KUKA KRL program: f1_Kuka_APT218T02S18.SRC

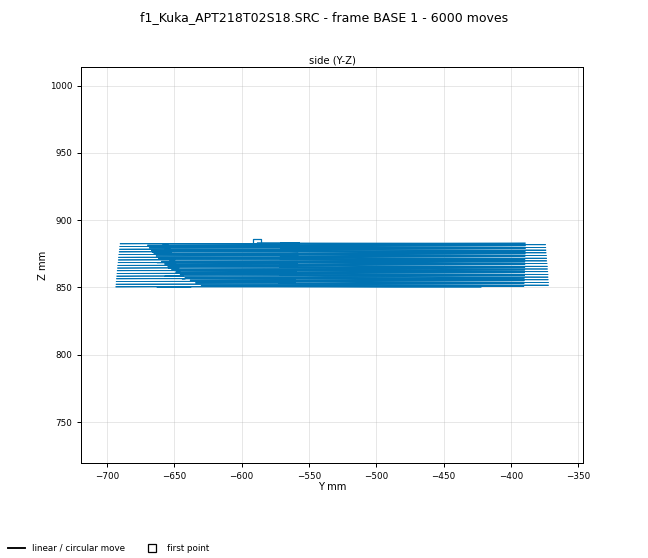
[picture p0: tool path of f1_Kuka_APT218T02S18.SRC in frame BASE 1, 6000 of 6001 moves have a stored position in this frame; points joined in program order, loops and branches not executed]
&ACCESS RVP
&REL 2
&PARAM TEMPLATE = C:\KRC\Roboter\Template\vorgabe
&PARAM EDITMASK = *
DEF f1_Kuka_APT218T02S18()


;FOLD INI;%{PE}%V3.2.0,%MKUKATPBASIS,%CINIT,%VCOMMON,%P
  ;FOLD BAS INI;%{E}%V3.2.0,%MKUKATPBASIS,%CINIT,%VINIT,%P
    GLOBAL INTERRUPT DECL 3 WHEN $STOPMESS==TRUE DO IR_STOPM ( )
    INTERRUPT ON 3
    BAS (#INITMOV,0 )
  ;ENDFOLD (BAS INI)
  ;FOLD USER INI;%{E}%V3.2.0,%MKUKATPUSER,%CINIT,%VINIT,%P
    ;Make your modifications here
  ;ENDFOLD (USER INI)
;ENDFOLD (INI)


;*** Make Null PTP Move
  PTP $pos_act

;*** Auto Load The Correct TOOL Data
  $tool=tool_data[2]

;*** Auto Load The Correct BASE Data
  $base=base_data[1]

  $ADVANCE = 5

;*** Restate Last Velocity
MMPM(30000.0)
SetRPM(8000)
LIN {X 0.122,Y -588.379,Z 883.406,A 0.000,B 0.000,C 90.000,E1 109.033} C_DIS
LIN {X -0.101,Y -579.806,Z 883.404,A 0.000,B 0.000,C 90.000,E1 108.671} C_DIS
LIN {X -0.188,Y -568.248,Z 883.402,A 0.000,B 0.000,C 90.000,E1 108.290} C_DIS
LIN {X -0.241,Y -564.785,Z 883.401,A 0.000,B 0.000,C 90.000,E1 108.181} C_DIS
LIN {X -0.107,Y -562.267,Z 883.400,A 0.000,B 0.000,C 90.000,E1 108.055} C_DIS
LIN {X 0.277,Y -559.252,Z 883.399,A 0.000,B 0.000,C 90.000,E1 107.819} C_DIS
LIN {X 0.169,Y -557.826,Z 883.398,A 0.000,B 0.000,C 90.000,E1 107.583} C_DIS
LIN {X -0.019,Y -557.157,Z 883.396,A 0.000,B 0.000,C 90.000,E1 107.221} C_DIS
LIN {X -0.140,Y -557.033,Z 883.393,A 0.000,B 0.000,C 90.000,E1 106.677} C_DIS
LIN {X 0.137,Y -558.022,Z 883.376,A 0.000,B 0.000,C 90.000,E1 103.592} C_DIS
LIN {X 0.043,Y -559.152,Z 883.365,A 0.000,B 0.000,C 90.000,E1 101.658} C_DIS
LIN {X -0.031,Y -560.530,Z 883.354,A 0.000,B 0.000,C 90.000,E1 99.726} C_DIS
LIN {X -0.015,Y -561.492,Z 883.346,A 0.000,B 0.000,C 90.000,E1 98.341} C_DIS
LIN {X 0.100,Y -562.358,Z 883.339,A 0.000,B 0.000,C 90.000,E1 96.947} C_DIS
LIN {X 0.092,Y -563.149,Z 883.331,A 0.000,B 0.000,C 90.000,E1 95.568} C_DIS
LIN {X 0.246,Y -563.909,Z 883.322,A 0.000,B 0.000,C 90.000,E1 93.898} C_DIS
LIN {X 0.231,Y -564.401,Z 883.314,A 0.000,B 0.000,C 90.000,E1 92.522} C_DIS
LIN {X -0.229,Y -564.932,Z 883.305,A 0.000,B 0.000,C 90.000,E1 90.917} C_DIS
LIN {X -0.237,Y -565.272,Z 883.297,A 0.000,B 0.000,C 90.000,E1 89.542} C_DIS
LIN {X -0.226,Y -565.571,Z 883.290,A 0.000,B 0.000,C 90.000,E1 88.165} C_DIS
LIN {X -0.093,Y -565.844,Z 883.281,A 0.000,B 0.000,C 90.000,E1 86.502} C_DIS
LIN {X -0.033,Y -566.089,Z 883.273,A 0.000,B 0.000,C 90.000,E1 85.122} C_DIS
LIN {X -0.274,Y -566.409,Z 883.262,A 0.000,B 0.000,C 90.000,E1 83.223} C_DIS
LIN {X -0.283,Y -566.973,Z 883.250,A 0.000,B 0.000,C 90.000,E1 81.027} C_DIS
LIN {X 0.107,Y -567.557,Z 883.241,A 0.000,B 0.000,C 90.000,E1 79.342} C_DIS
LIN {X 0.241,Y -568.440,Z 883.230,A 0.000,B 0.000,C 90.000,E1 77.409} C_DIS
LIN {X 0.029,Y -569.048,Z 883.223,A 0.000,B 0.000,C 90.000,E1 76.061} C_DIS
LIN {X -0.040,Y -569.635,Z 883.215,A 0.000,B 0.000,C 90.000,E1 74.700} C_DIS
LIN {X -0.120,Y -570.012,Z 883.209,A 0.000,B 0.000,C 90.000,E1 73.614} C_DIS
LIN {X 0.162,Y -570.430,Z 883.200,A 0.000,B 0.000,C 90.000,E1 71.945} C_DIS
LIN {X 0.102,Y -570.623,Z 883.194,A 0.000,B 0.000,C 90.000,E1 70.859} C_DIS
LIN {X 0.237,Y -570.806,Z 883.188,A 0.000,B 0.000,C 90.000,E1 69.752} C_DIS
LIN {X -0.001,Y -570.993,Z 883.176,A 0.000,B 0.000,C 90.000,E1 67.592} C_DIS
LIN {X 0.141,Y -571.068,Z 883.169,A 0.000,B 0.000,C 90.000,E1 66.485} C_DIS
LIN {X 0.169,Y -571.046,Z 883.160,A 0.000,B 0.000,C 90.000,E1 64.845} C_DIS
LIN {X 0.190,Y -570.924,Z 883.151,A 0.000,B 0.000,C 90.000,E1 63.204} C_DIS
LIN {X -0.057,Y -570.579,Z 883.142,A 0.000,B 0.000,C 90.000,E1 61.591} C_DIS
LIN {X 0.309,Y -570.340,Z 883.136,A 0.000,B 0.000,C 90.000,E1 60.461} C_DIS
LIN {X 0.073,Y -570.058,Z 883.132,A 0.000,B 0.000,C 90.000,E1 59.665} C_DIS
LIN {X -0.113,Y -569.130,Z 883.122,A 0.000,B 0.000,C 90.000,E1 58.043} C_DIS
LIN {X 0.113,Y -568.574,Z 883.118,A 0.000,B 0.000,C 90.000,E1 57.199} C_DIS
LIN {X 0.155,Y -567.877,Z 883.113,A 0.000,B 0.000,C 90.000,E1 56.373} C_DIS
LIN {X -0.158,Y -566.857,Z 883.107,A 0.000,B 0.000,C 90.000,E1 55.308} C_DIS
LIN {X -0.016,Y -565.616,Z 883.101,A 0.000,B 0.000,C 90.000,E1 54.196} C_DIS
LIN {X -0.352,Y -564.093,Z 883.095,A 0.000,B 0.000,C 90.000,E1 53.130} C_DIS
LIN {X -0.028,Y -562.837,Z 883.090,A 0.000,B 0.000,C 90.000,E1 52.271} C_DIS
LIN {X -0.161,Y -561.473,Z 883.086,A 0.000,B 0.000,C 90.000,E1 51.457} C_DIS
LIN {X 0.127,Y -559.875,Z 883.081,A 0.000,B 0.000,C 90.000,E1 50.598} C_DIS
LIN {X -0.124,Y -558.727,Z 883.078,A 0.000,B 0.000,C 90.000,E1 50.070} C_DIS
LIN {X 0.061,Y -556.766,Z 883.074,A 0.000,B 0.000,C 90.000,E1 49.218} C_DIS
LIN {X 0.296,Y -553.482,Z 883.067,A 0.000,B 0.000,C 90.000,E1 48.081} C_DIS
LIN {X 0.004,Y -551.691,Z 883.064,A 0.000,B 0.000,C 90.000,E1 47.553} C_DIS
LIN {X 0.113,Y -548.706,Z 883.060,A 0.000,B 0.000,C 90.000,E1 46.701} C_DIS
LIN {X -0.205,Y -545.511,Z 883.055,A 0.000,B 0.000,C 90.000,E1 45.891} C_DIS
LIN {X 0.217,Y -541.967,Z 883.050,A 0.000,B 0.000,C 90.000,E1 45.000} C_DIS
LIN {X 0.018,Y -538.556,Z 883.046,A 0.000,B 0.000,C 90.000,E1 44.312} C_DIS
LIN {X -0.203,Y -534.722,Z 883.042,A 0.000,B 0.000,C 90.000,E1 43.623} C_DIS
LIN {X -0.090,Y -530.576,Z 883.038,A 0.000,B 0.000,C 90.000,E1 42.894} C_DIS
LIN {X 0.211,Y -527.049,Z 883.035,A 0.000,B 0.000,C 90.000,E1 42.285} C_DIS
LIN {X 0.045,Y -521.421,Z 883.030,A 0.000,B 0.000,C 90.000,E1 41.434} C_DIS
LIN {X 0.007,Y -513.993,Z 883.025,A 0.000,B 0.000,C 90.000,E1 40.415} C_DIS
LIN {X 0.301,Y -508.245,Z 883.021,A 0.000,B 0.000,C 90.000,E1 39.644} C_DIS
LIN {X 0.213,Y -501.947,Z 883.016,A 0.000,B 0.000,C 90.000,E1 38.910} C_DIS
LIN {X 0.220,Y -497.947,Z 883.014,A 0.000,B 0.000,C 90.000,E1 38.463} C_DIS
LIN {X -0.149,Y -489.660,Z 883.009,A 0.000,B 0.000,C 90.000,E1 37.649} C_DIS
LIN {X -0.010,Y -483.974,Z 883.006,A 0.000,B 0.000,C 90.000,E1 37.076} C_DIS
LIN {X 0.171,Y -476.519,Z 883.002,A 0.000,B 0.000,C 90.000,E1 36.377} C_DIS
LIN {X -0.193,Y -466.025,Z 882.997,A 0.000,B 0.000,C 90.000,E1 35.518} C_DIS
LIN {X -0.045,Y -458.299,Z 882.994,A 0.000,B 0.000,C 90.000,E1 34.865} C_DIS
LIN {X -0.104,Y -450.565,Z 882.990,A 0.000,B 0.000,C 90.000,E1 34.246} C_DIS
LIN {X 0.184,Y -435.026,Z 882.983,A 0.000,B 0.000,C 90.000,E1 32.959} C_DIS
LIN {X -0.153,Y -418.321,Z 882.975,A 0.000,B 0.000,C 90.000,E1 31.592} C_DIS
LIN {X -0.172,Y -404.709,Z 882.968,A 0.000,B 0.000,C 90.000,E1 30.335} C_DIS
LIN {X 0.006,Y -397.858,Z 882.964,A 0.000,B 0.000,C 90.000,E1 29.589} C_DIS
LIN {X -0.089,Y -395.270,Z 882.963,A 0.000,B 0.000,C 90.000,E1 29.283} C_DIS
LIN {X 0.077,Y -393.465,Z 882.961,A 0.000,B 0.000,C 90.000,E1 28.999} C_DIS
LIN {X 0.060,Y -391.088,Z 882.958,A 0.000,B 0.000,C 90.000,E1 28.487} C_DIS
LIN {X -0.130,Y -390.109,Z 882.956,A 0.000,B 0.000,C 90.000,E1 28.153} C_DIS
LIN {X -0.125,Y -389.776,Z 882.955,A 0.000,B 0.000,C 90.000,E1 27.975} C_DIS
LIN {X -0.066,Y -389.241,Z 882.952,A 0.000,B 0.000,C 90.000,E1 27.436} C_DIS
LIN {X -0.178,Y -389.129,Z 882.948,A 0.000,B 0.000,C 90.000,E1 26.744} C_DIS
LIN {X -0.114,Y -390.003,Z 882.939,A 0.000,B 0.000,C 90.000,E1 24.951} C_DIS
LIN {X 0.108,Y -392.719,Z 882.921,A 0.000,B 0.000,C 90.000,E1 21.716} C_DIS
LIN {X -0.171,Y -394.920,Z 882.909,A 0.000,B 0.000,C 90.000,E1 19.631} C_DIS
LIN {X -0.095,Y -397.735,Z 882.895,A 0.000,B 0.000,C 90.000,E1 17.149} C_DIS
LIN {X 0.184,Y -401.298,Z 882.880,A 0.000,B 0.000,C 90.000,E1 14.300} C_DIS
LIN {X -0.001,Y -405.149,Z 882.864,A 0.000,B 0.000,C 90.000,E1 11.535} C_DIS
LIN {X 0.084,Y -408.893,Z 882.851,A 0.000,B 0.000,C 90.000,E1 9.095} C_DIS
LIN {X -0.156,Y -413.579,Z 882.835,A 0.000,B 0.000,C 90.000,E1 6.372} C_DIS
LIN {X 0.009,Y -418.079,Z 882.822,A 0.000,B 0.000,C 90.000,E1 3.955} C_DIS
LIN {X -0.043,Y -425.252,Z 882.803,A 0.000,B 0.000,C 90.000,E1 0.573} C_DIS
LIN {X -0.010,Y -430.285,Z 882.791,A 0.000,B 0.000,C 90.000,E1 358.453} C_DIS
LIN {X -0.159,Y -437.144,Z 882.777,A 0.000,B 0.000,C 90.000,E1 355.812} C_DIS
LIN {X 0.066,Y -439.313,Z 882.773,A 0.000,B 0.000,C 90.000,E1 355.122} C_DIS
LIN {X 0.067,Y -442.262,Z 882.770,A 0.000,B 0.000,C 90.000,E1 354.546} C_DIS
LIN {X 0.180,Y -444.846,Z 882.768,A 0.000,B 0.000,C 90.000,E1 354.204} C_DIS
LIN {X 0.121,Y -449.563,Z 882.766,A 0.000,B 0.000,C 90.000,E1 353.856} C_DIS
LIN {X 0.062,Y -455.330,Z 882.764,A 0.000,B 0.000,C 90.000,E1 353.571} C_DIS
LIN {X -0.058,Y -468.891,Z 882.761,A 0.000,B 0.000,C 90.000,E1 352.996} C_DIS
LIN {X -0.002,Y -477.211,Z 882.759,A 0.000,B 0.000,C 90.000,E1 352.591} C_DIS
LIN {X 0.067,Y -483.618,Z 882.757,A 0.000,B 0.000,C 90.000,E1 352.243} C_DIS
LIN {X 0.101,Y -491.818,Z 882.754,A 0.000,B 0.000,C 90.000,E1 351.781} C_DIS
LIN {X 0.245,Y -501.546,Z 882.751,A 0.000,B 0.000,C 90.000,E1 351.197} C_DIS
LIN {X 0.051,Y -510.970,Z 882.748,A 0.000,B 0.000,C 90.000,E1 350.622} C_DIS
LIN {X 0.091,Y -518.862,Z 882.745,A 0.000,B 0.000,C 90.000,E1 350.095} C_DIS
LIN {X 0.016,Y -526.453,Z 882.742,A 0.000,B 0.000,C 90.000,E1 349.567} C_DIS
LIN {X 0.149,Y -532.466,Z 882.740,A 0.000,B 0.000,C 90.000,E1 349.106} C_DIS
LIN {X 0.151,Y -539.715,Z 882.736,A 0.000,B 0.000,C 90.000,E1 348.522} C_DIS
LIN {X -0.009,Y -546.525,Z 882.733,A 0.000,B 0.000,C 90.000,E1 347.937} C_DIS
LIN {X -0.075,Y -554.603,Z 882.729,A 0.000,B 0.000,C 90.000,E1 347.173} C_DIS
LIN {X -0.137,Y -561.000,Z 882.725,A 0.000,B 0.000,C 90.000,E1 346.520} C_DIS
LIN {X -0.028,Y -567.119,Z 882.721,A 0.000,B 0.000,C 90.000,E1 345.825} C_DIS
LIN {X -0.095,Y -571.726,Z 882.718,A 0.000,B 0.000,C 90.000,E1 345.283} C_DIS
LIN {X -0.175,Y -579.173,Z 882.713,A 0.000,B 0.000,C 90.000,E1 344.338} C_DIS
LIN {X 0.159,Y -584.078,Z 882.709,A 0.000,B 0.000,C 90.000,E1 343.630} C_DIS
LIN {X -0.176,Y -590.395,Z 882.704,A 0.000,B 0.000,C 90.000,E1 342.725} C_DIS
LIN {X 0.070,Y -597.021,Z 882.698,A 0.000,B 0.000,C 90.000,E1 341.638} C_DIS
LIN {X -0.155,Y -603.051,Z 882.692,A 0.000,B 0.000,C 90.000,E1 340.604} C_DIS
LIN {X -0.235,Y -607.309,Z 882.688,A 0.000,B 0.000,C 90.000,E1 339.826} C_DIS
LIN {X -0.158,Y -614.014,Z 882.681,A 0.000,B 0.000,C 90.000,E1 338.518} C_DIS
LIN {X -0.159,Y -618.460,Z 882.676,A 0.000,B 0.000,C 90.000,E1 337.614} C_DIS
LIN {X 0.116,Y -623.243,Z 882.670,A 0.000,B 0.000,C 90.000,E1 336.561} C_DIS
LIN {X 0.131,Y -627.747,Z 882.664,A 0.000,B 0.000,C 90.000,E1 335.537} C_DIS
LIN {X -0.049,Y -631.918,Z 882.659,A 0.000,B 0.000,C 90.000,E1 334.537} C_DIS
LIN {X 0.096,Y -635.794,Z 882.653,A 0.000,B 0.000,C 90.000,E1 333.512} C_DIS
LIN {X 0.293,Y -639.458,Z 882.647,A 0.000,B 0.000,C 90.000,E1 332.487} C_DIS
LIN {X 0.036,Y -643.618,Z 882.640,A 0.000,B 0.000,C 90.000,E1 331.257} C_DIS
LIN {X 0.237,Y -648.155,Z 882.632,A 0.000,B 0.000,C 90.000,E1 329.744} C_DIS
LIN {X 0.258,Y -650.302,Z 882.628,A 0.000,B 0.000,C 90.000,E1 328.997} C_DIS
LIN {X -0.065,Y -653.728,Z 882.621,A 0.000,B 0.000,C 90.000,E1 327.788} C_DIS
LIN {X 0.110,Y -656.122,Z 882.616,A 0.000,B 0.000,C 90.000,E1 326.786} C_DIS
LIN {X 0.128,Y -658.310,Z 882.610,A 0.000,B 0.000,C 90.000,E1 325.801} C_DIS
LIN {X 0.183,Y -660.174,Z 882.605,A 0.000,B 0.000,C 90.000,E1 324.815} C_DIS
LIN {X 0.265,Y -661.759,Z 882.599,A 0.000,B 0.000,C 90.000,E1 323.829} C_DIS
LIN {X 0.363,Y -663.180,Z 882.594,A 0.000,B 0.000,C 90.000,E1 322.844} C_DIS
LIN {X -0.023,Y -664.153,Z 882.590,A 0.000,B 0.000,C 90.000,E1 322.145} C_DIS
LIN {X -0.040,Y -665.507,Z 882.583,A 0.000,B 0.000,C 90.000,E1 320.928} C_DIS
LIN {X 0.065,Y -666.817,Z 882.576,A 0.000,B 0.000,C 90.000,E1 319.703} C_DIS
LIN {X 0.103,Y -668.353,Z 882.568,A 0.000,B 0.000,C 90.000,E1 318.243} C_DIS
LIN {X -0.324,Y -669.643,Z 882.561,A 0.000,B 0.000,C 90.000,E1 317.067} C_DIS
LIN {X 0.217,Y -670.951,Z 882.555,A 0.000,B 0.000,C 90.000,E1 315.810} C_DIS
LIN {X 0.299,Y -672.265,Z 882.548,A 0.000,B 0.000,C 90.000,E1 314.595} C_DIS
LIN {X -0.022,Y -673.927,Z 882.539,A 0.000,B 0.000,C 90.000,E1 312.933} C_DIS
LIN {X -0.363,Y -675.092,Z 882.532,A 0.000,B 0.000,C 90.000,E1 311.757} C_DIS
LIN {X -0.208,Y -675.929,Z 882.526,A 0.000,B 0.000,C 90.000,E1 310.782} C_DIS
LIN {X 0.118,Y -677.365,Z 882.517,A 0.000,B 0.000,C 90.000,E1 309.072} C_DIS
LIN {X -0.084,Y -678.489,Z 882.509,A 0.000,B 0.000,C 90.000,E1 307.649} C_DIS
LIN {X -0.163,Y -679.400,Z 882.503,A 0.000,B 0.000,C 90.000,E1 306.457} C_DIS
LIN {X 0.172,Y -680.053,Z 882.497,A 0.000,B 0.000,C 90.000,E1 305.471} C_DIS
LIN {X 0.303,Y -681.034,Z 882.488,A 0.000,B 0.000,C 90.000,E1 303.785} C_DIS
LIN {X 0.448,Y -681.993,Z 882.480,A 0.000,B 0.000,C 90.000,E1 302.339} C_DIS
LIN {X 0.060,Y -683.481,Z 882.469,A 0.000,B 0.000,C 90.000,E1 300.463} C_DIS
LIN {X 0.181,Y -685.412,Z 882.457,A 0.000,B 0.000,C 90.000,E1 298.309} C_DIS
LIN {X 0.129,Y -687.513,Z 882.447,A 0.000,B 0.000,C 90.000,E1 296.411} C_DIS
LIN {X 0.345,Y -688.947,Z 882.440,A 0.000,B 0.000,C 90.000,E1 295.207} C_DIS
LIN {X 0.069,Y -689.832,Z 882.435,A 0.000,B 0.000,C 90.000,E1 294.283} C_DIS
LIN {X 0.135,Y -690.317,Z 882.431,A 0.000,B 0.000,C 90.000,E1 293.567} C_DIS
LIN {X 0.092,Y -690.368,Z 882.430,A 0.000,B 0.000,C 90.000,E1 293.334} C_DIS
LIN {X -0.350,Y -690.024,Z 882.427,A 0.000,B 0.000,C 90.000,E1 292.898} C_DIS
LIN {X -0.120,Y -689.571,Z 882.426,A 0.000,B 0.000,C 90.000,E1 292.642} C_DIS
LIN {X 0.072,Y -687.982,Z 882.423,A 0.000,B 0.000,C 90.000,E1 292.153} C_DIS
LIN {X 0.183,Y -687.443,Z 882.422,A 0.000,B 0.000,C 90.000,E1 292.025} C_DIS
LIN {X 0.294,Y -686.610,Z 882.422,A 0.000,B 0.000,C 90.000,E1 291.897} C_DIS
LIN {X 0.254,Y -684.050,Z 882.421,A 0.000,B 0.000,C 90.000,E1 291.663} C_DIS
LIN {X -0.185,Y -682.758,Z 882.420,A 0.000,B 0.000,C 90.000,E1 291.589} C_DIS
LIN {X 0.055,Y -679.828,Z 882.419,A 0.000,B 0.000,C 90.000,E1 291.354} C_DIS
LIN {X -0.284,Y -677.735,Z 882.418,A 0.000,B 0.000,C 90.000,E1 291.280} C_DIS
LIN {X 0.307,Y -669.422,Z 882.417,A 0.000,B 0.000,C 90.000,E1 290.972} C_DIS
LIN {X 0.039,Y -661.806,Z 882.416,A 0.000,B 0.000,C 90.000,E1 290.791} C_DIS
LIN {X -0.137,Y -660.012,Z 882.415,A 0.000,B 0.000,C 90.000,E1 290.737} C_DIS
LIN {X -0.188,Y -655.626,Z 882.414,A 0.000,B 0.000,C 90.000,E1 290.536} C_DIS
LIN {X 0.371,Y -655.532,Z 882.414,A 0.000,B 0.000,C 90.000,E1 290.482} C_DIS
LIN {X -0.298,Y -654.580,Z 882.413,A 0.000,B 0.000,C 90.000,E1 290.429} C_DIS
LIN {X -0.342,Y -654.560,Z 882.413,A 0.000,B 0.000,C 90.000,E1 290.429} C_DIS
LIN {X 0.106,Y -654.455,Z 882.412,A 0.000,B 0.000,C 90.000,E1 290.174} C_DIS
LIN {X -0.068,Y -655.646,Z 882.410,A 0.000,B 0.000,C 90.000,E1 289.758} C_DIS
LIN {X 0.128,Y -658.793,Z 882.406,A 0.000,B 0.000,C 90.000,E1 289.087} C_DIS
LIN {X 0.056,Y -665.349,Z 882.399,A 0.000,B 0.000,C 90.000,E1 287.873} C_DIS
LIN {X -0.010,Y -668.755,Z 882.395,A 0.000,B 0.000,C 90.000,E1 287.149} C_DIS
LIN {X -0.238,Y -671.708,Z 882.391,A 0.000,B 0.000,C 90.000,E1 286.441} C_DIS
LIN {X -0.184,Y -673.408,Z 882.389,A 0.000,B 0.000,C 90.000,E1 285.953} C_DIS
LIN {X 0.287,Y -675.387,Z 882.385,A 0.000,B 0.000,C 90.000,E1 285.190} C_DIS
LIN {X 0.134,Y -676.960,Z 882.381,A 0.000,B 0.000,C 90.000,E1 284.481} C_DIS
LIN {X -0.003,Y -678.229,Z 882.377,A 0.000,B 0.000,C 90.000,E1 283.772} C_DIS
LIN {X -0.129,Y -679.262,Z 882.373,A 0.000,B 0.000,C 90.000,E1 283.063} C_DIS
LIN {X -0.249,Y -679.961,Z 882.369,A 0.000,B 0.000,C 90.000,E1 282.355} C_DIS
LIN {X 0.338,Y -680.308,Z 882.366,A 0.000,B 0.000,C 90.000,E1 281.827} C_DIS
LIN {X 0.125,Y -680.466,Z 882.363,A 0.000,B 0.000,C 90.000,E1 281.366} C_DIS
LIN {X 0.008,Y -680.140,Z 882.359,A 0.000,B 0.000,C 90.000,E1 280.658} C_DIS
LIN {X -0.199,Y -679.695,Z 882.357,A 0.000,B 0.000,C 90.000,E1 280.197} C_DIS
LIN {X -0.287,Y -678.957,Z 882.354,A 0.000,B 0.000,C 90.000,E1 279.726} C_DIS
LIN {X 0.173,Y -677.860,Z 882.351,A 0.000,B 0.000,C 90.000,E1 279.208} C_DIS
LIN {X -0.038,Y -676.482,Z 882.349,A 0.000,B 0.000,C 90.000,E1 278.746} C_DIS
LIN {X -0.096,Y -675.722,Z 882.347,A 0.000,B 0.000,C 90.000,E1 278.511} C_DIS
LIN {X -0.318,Y -673.947,Z 882.345,A 0.000,B 0.000,C 90.000,E1 278.049} C_DIS
LIN {X 0.118,Y -671.850,Z 882.342,A 0.000,B 0.000,C 90.000,E1 277.530} C_DIS
LIN {X -0.126,Y -668.852,Z 882.339,A 0.000,B 0.000,C 90.000,E1 276.947} C_DIS
LIN {X 0.181,Y -665.352,Z 882.335,A 0.000,B 0.000,C 90.000,E1 276.315} C_DIS
LIN {X -0.108,Y -662.244,Z 882.333,A 0.000,B 0.000,C 90.000,E1 275.853} C_DIS
LIN {X 0.239,Y -658.650,Z 882.330,A 0.000,B 0.000,C 90.000,E1 275.334} C_DIS
LIN {X -0.197,Y -653.477,Z 882.326,A 0.000,B 0.000,C 90.000,E1 274.759} C_DIS
LIN {X 0.058,Y -648.780,Z 882.324,A 0.000,B 0.000,C 90.000,E1 274.245} C_DIS
LIN {X -0.202,Y -643.723,Z 882.321,A 0.000,B 0.000,C 90.000,E1 273.784} C_DIS
LIN {X 0.298,Y -637.049,Z 882.318,A 0.000,B 0.000,C 90.000,E1 273.154} C_DIS
LIN {X -0.158,Y -631.515,Z 882.315,A 0.000,B 0.000,C 90.000,E1 272.751} C_DIS
LIN {X -0.289,Y -623.990,Z 882.312,A 0.000,B 0.000,C 90.000,E1 272.236} C_DIS
LIN {X -0.088,Y -617.778,Z 882.310,A 0.000,B 0.000,C 90.000,E1 271.835} C_DIS
LIN {X -0.203,Y -611.264,Z 882.308,A 0.000,B 0.000,C 90.000,E1 271.489} C_DIS
LIN {X -0.011,Y -604.489,Z 882.306,A 0.000,B 0.000,C 90.000,E1 271.146} C_DIS
LIN {X -0.109,Y -597.612,Z 882.305,A 0.000,B 0.000,C 90.000,E1 270.859} C_DIS
LIN {X 0.162,Y -590.393,Z 882.303,A 0.000,B 0.000,C 90.000,E1 270.573} C_DIS
LIN {X -0.278,Y -582.943,Z 882.302,A 0.000,B 0.000,C 90.000,E1 270.401} C_DIS
LIN {X 0.038,Y -577.504,Z 882.301,A 0.000,B 0.000,C 90.000,E1 270.229} C_DIS
LIN {X -0.107,Y -571.034,Z 882.301,A 0.000,B 0.000,C 90.000,E1 270.115} C_DIS
LIN {X 0.195,Y -563.729,Z 882.300,A 0.000,B 0.000,C 90.000,E1 270.000} C_DIS
LIN {X -0.009,Y -552.379,Z 882.300,A 0.000,B 0.000,C 90.000,E1 269.943} C_DIS
LIN {X -0.195,Y -549.486,Z 882.299,A 0.000,B 0.000,C 90.000,E1 269.885} C_DIS
LIN {X -0.224,Y -549.437,Z 882.299,A 0.000,B 0.000,C 90.000,E1 269.885} C_DIS
LIN {X 0.068,Y -546.726,Z 882.298,A 0.000,B 0.000,C 90.000,E1 269.542} C_DIS
LIN {X -0.056,Y -546.333,Z 882.297,A 0.000,B 0.000,C 90.000,E1 269.484} C_DIS
LIN {X 0.115,Y -545.774,Z 882.296,A 0.000,B 0.000,C 90.000,E1 269.255} C_DIS
LIN {X -0.249,Y -544.841,Z 882.293,A 0.000,B 0.000,C 90.000,E1 268.740} C_DIS
LIN {X 0.254,Y -541.460,Z 882.271,A 0.000,B 0.000,C 90.000,E1 264.723} C_DIS
LIN {X -0.067,Y -540.539,Z 882.263,A 0.000,B 0.000,C 90.000,E1 263.337} C_DIS
LIN {X 0.066,Y -539.640,Z 882.257,A 0.000,B 0.000,C 90.000,E1 262.186} C_DIS
LIN {X -0.210,Y -538.259,Z 882.249,A 0.000,B 0.000,C 90.000,E1 260.792} C_DIS
LIN {X 0.080,Y -536.471,Z 882.239,A 0.000,B 0.000,C 90.000,E1 259.050} C_DIS
LIN {X -0.153,Y -534.963,Z 882.231,A 0.000,B 0.000,C 90.000,E1 257.645} C_DIS
LIN {X 0.177,Y -533.606,Z 882.225,A 0.000,B 0.000,C 90.000,E1 256.464} C_DIS
LIN {X 0.052,Y -531.429,Z 882.215,A 0.000,B 0.000,C 90.000,E1 254.755} C_DIS
LIN {X 0.164,Y -529.324,Z 882.206,A 0.000,B 0.000,C 90.000,E1 253.015} C_DIS
LIN {X 0.059,Y -527.638,Z 882.198,A 0.000,B 0.000,C 90.000,E1 251.583} C_DIS
LIN {X -0.248,Y -525.386,Z 882.188,A 0.000,B 0.000,C 90.000,E1 249.880} C_DIS
LIN {X -0.090,Y -523.463,Z 882.180,A 0.000,B 0.000,C 90.000,E1 248.411} C_DIS
LIN {X 0.222,Y -521.303,Z 882.172,A 0.000,B 0.000,C 90.000,E1 246.922} C_DIS
LIN {X -0.129,Y -519.547,Z 882.165,A 0.000,B 0.000,C 90.000,E1 245.793} C_DIS
LIN {X -0.148,Y -517.318,Z 882.157,A 0.000,B 0.000,C 90.000,E1 244.332} C_DIS
LIN {X 0.006,Y -515.924,Z 882.152,A 0.000,B 0.000,C 90.000,E1 243.435} C_DIS
LIN {X -0.198,Y -513.885,Z 882.146,A 0.000,B 0.000,C 90.000,E1 242.281} C_DIS
LIN {X -0.095,Y -511.318,Z 882.138,A 0.000,B 0.000,C 90.000,E1 240.795} C_DIS
LIN {X -0.237,Y -508.789,Z 882.130,A 0.000,B 0.000,C 90.000,E1 239.331} C_DIS
LIN {X -0.051,Y -506.637,Z 882.123,A 0.000,B 0.000,C 90.000,E1 238.122} C_DIS
LIN {X -0.216,Y -504.969,Z 882.118,A 0.000,B 0.000,C 90.000,E1 237.248} C_DIS
LIN {X 0.182,Y -502.556,Z 882.111,A 0.000,B 0.000,C 90.000,E1 236.008} C_DIS
LIN {X 0.247,Y -500.622,Z 882.106,A 0.000,B 0.000,C 90.000,E1 235.102} C_DIS
LIN {X -0.227,Y -495.716,Z 882.095,A 0.000,B 0.000,C 90.000,E1 233.050} C_DIS
LIN {X -0.233,Y -492.184,Z 882.086,A 0.000,B 0.000,C 90.000,E1 231.537} C_DIS
LIN {X 0.003,Y -490.085,Z 882.081,A 0.000,B 0.000,C 90.000,E1 230.598} C_DIS
LIN {X -0.188,Y -486.633,Z 882.073,A 0.000,B 0.000,C 90.000,E1 229.094} C_DIS
LIN {X 0.066,Y -483.856,Z 882.066,A 0.000,B 0.000,C 90.000,E1 227.838} C_DIS
LIN {X 0.209,Y -479.862,Z 882.056,A 0.000,B 0.000,C 90.000,E1 225.972} C_DIS
LIN {X 0.240,Y -475.684,Z 882.045,A 0.000,B 0.000,C 90.000,E1 224.109} C_DIS
LIN {X -0.155,Y -471.504,Z 882.035,A 0.000,B 0.000,C 90.000,E1 222.285} C_DIS
LIN {X -0.019,Y -467.983,Z 882.026,A 0.000,B 0.000,C 90.000,E1 220.701} C_DIS
LIN {X -0.005,Y -465.299,Z 882.019,A 0.000,B 0.000,C 90.000,E1 219.439} C_DIS
LIN {X 0.119,Y -461.226,Z 882.009,A 0.000,B 0.000,C 90.000,E1 217.523} C_DIS
LIN {X 0.121,Y -457.905,Z 882.000,A 0.000,B 0.000,C 90.000,E1 215.931} C_DIS
LIN {X -0.121,Y -453.851,Z 881.989,A 0.000,B 0.000,C 90.000,E1 214.040} C_DIS
LIN {X -0.123,Y -451.046,Z 881.982,A 0.000,B 0.000,C 90.000,E1 212.752} C_DIS
LIN {X -0.165,Y -448.371,Z 881.975,A 0.000,B 0.000,C 90.000,E1 211.465} C_DIS
LIN {X 0.101,Y -443.471,Z 881.962,A 0.000,B 0.000,C 90.000,E1 209.155} C_DIS
LIN {X 0.101,Y -440.578,Z 881.955,A 0.000,B 0.000,C 90.000,E1 207.847} C_DIS
LIN {X -0.098,Y -436.206,Z 881.944,A 0.000,B 0.000,C 90.000,E1 205.899} C_DIS
LIN {X 0.188,Y -432.714,Z 881.935,A 0.000,B 0.000,C 90.000,E1 204.207} C_DIS
LIN {X 0.029,Y -429.943,Z 881.927,A 0.000,B 0.000,C 90.000,E1 202.898} C_DIS
LIN {X 0.024,Y -425.097,Z 881.914,A 0.000,B 0.000,C 90.000,E1 200.556} C_DIS
LIN {X -0.226,Y -421.712,Z 881.905,A 0.000,B 0.000,C 90.000,E1 198.906} C_DIS
LIN {X -0.117,Y -417.612,Z 881.894,A 0.000,B 0.000,C 90.000,E1 196.858} C_DIS
LIN {X -0.197,Y -412.761,Z 881.880,A 0.000,B 0.000,C 90.000,E1 194.481} C_DIS
LIN {X 0.147,Y -409.461,Z 881.871,A 0.000,B 0.000,C 90.000,E1 192.715} C_DIS
LIN {X 0.017,Y -406.102,Z 881.861,A 0.000,B 0.000,C 90.000,E1 191.007} C_DIS
LIN {X 0.054,Y -403.406,Z 881.854,A 0.000,B 0.000,C 90.000,E1 189.613} C_DIS
LIN {X -0.028,Y -399.139,Z 881.842,A 0.000,B 0.000,C 90.000,E1 187.530} C_DIS
LIN {X -0.062,Y -392.690,Z 881.822,A 0.000,B 0.000,C 90.000,E1 184.012} C_DIS
LIN {X 0.086,Y -388.307,Z 881.806,A 0.000,B 0.000,C 90.000,E1 181.146} C_DIS
LIN {X 0.004,Y -385.723,Z 881.797,A 0.000,B 0.000,C 90.000,E1 179.370} C_DIS
LIN {X -0.124,Y -383.051,Z 881.787,A 0.000,B 0.000,C 90.000,E1 177.593} C_DIS
LIN {X 0.096,Y -380.292,Z 881.777,A 0.000,B 0.000,C 90.000,E1 175.755} C_DIS
LIN {X 0.045,Y -375.566,Z 881.756,A 0.000,B 0.000,C 90.000,E1 172.129} C_DIS
LIN {X -0.027,Y -374.541,Z 881.748,A 0.000,B 0.000,C 90.000,E1 170.679} C_DIS
LIN {X -0.140,Y -374.328,Z 881.746,A 0.000,B 0.000,C 90.000,E1 170.330} C_DIS
LIN {X -0.047,Y -374.214,Z 881.740,A 0.000,B 0.000,C 90.000,E1 169.218} C_DIS
LIN {X 0.089,Y -374.508,Z 881.736,A 0.000,B 0.000,C 90.000,E1 168.465} C_DIS
LIN {X -0.065,Y -375.254,Z 881.732,A 0.000,B 0.000,C 90.000,E1 167.757} C_DIS
LIN {X 0.157,Y -376.558,Z 881.728,A 0.000,B 0.000,C 90.000,E1 166.992} C_DIS
LIN {X 0.044,Y -377.457,Z 881.726,A 0.000,B 0.000,C 90.000,E1 166.645} C_DIS
LIN {X -0.086,Y -380.023,Z 881.722,A 0.000,B 0.000,C 90.000,E1 165.936} C_DIS
LIN {X 0.127,Y -382.241,Z 881.719,A 0.000,B 0.000,C 90.000,E1 165.463} C_DIS
LIN {X -0.077,Y -384.997,Z 881.717,A 0.000,B 0.000,C 90.000,E1 165.102} C_DIS
LIN {X -0.169,Y -388.168,Z 881.715,A 0.000,B 0.000,C 90.000,E1 164.755} C_DIS
LIN {X 0.115,Y -391.902,Z 881.713,A 0.000,B 0.000,C 90.000,E1 164.393} C_DIS
LIN {X 0.097,Y -395.132,Z 881.712,A 0.000,B 0.000,C 90.000,E1 164.157} C_DIS
LIN {X -0.133,Y -400.993,Z 881.710,A 0.000,B 0.000,C 90.000,E1 163.850} C_DIS
LIN {X 0.060,Y -409.802,Z 881.708,A 0.000,B 0.000,C 90.000,E1 163.378} C_DIS
LIN {X 0.095,Y -416.536,Z 881.706,A 0.000,B 0.000,C 90.000,E1 163.015} C_DIS
LIN {X -0.034,Y -422.901,Z 881.704,A 0.000,B 0.000,C 90.000,E1 162.653} C_DIS
LIN {X 0.213,Y -426.048,Z 881.703,A 0.000,B 0.000,C 90.000,E1 162.417} C_DIS
LIN {X 0.068,Y -435.487,Z 881.699,A 0.000,B 0.000,C 90.000,E1 161.764} C_DIS
LIN {X 0.162,Y -441.747,Z 881.696,A 0.000,B 0.000,C 90.000,E1 161.275} C_DIS
LIN {X -0.058,Y -450.861,Z 881.692,A 0.000,B 0.000,C 90.000,E1 160.550} C_DIS
LIN {X -0.125,Y -459.764,Z 881.688,A 0.000,B 0.000,C 90.000,E1 159.752} C_DIS
LIN {X -0.057,Y -468.140,Z 881.683,A 0.000,B 0.000,C 90.000,E1 158.901} C_DIS
LIN {X 0.190,Y -477.730,Z 881.677,A 0.000,B 0.000,C 90.000,E1 157.847} C_DIS
LIN {X 0.132,Y -484.228,Z 881.673,A 0.000,B 0.000,C 90.000,E1 157.102} C_DIS
LIN {X 0.167,Y -489.171,Z 881.669,A 0.000,B 0.000,C 90.000,E1 156.485} C_DIS
LIN {X 0.164,Y -491.437,Z 881.668,A 0.000,B 0.000,C 90.000,E1 156.230} C_DIS
LIN {X 0.126,Y -499.450,Z 881.662,A 0.000,B 0.000,C 90.000,E1 155.177} C_DIS
LIN {X -0.181,Y -505.003,Z 881.658,A 0.000,B 0.000,C 90.000,E1 154.460} C_DIS
LIN {X -0.156,Y -511.378,Z 881.653,A 0.000,B 0.000,C 90.000,E1 153.563} C_DIS
LIN {X -0.058,Y -517.390,Z 881.648,A 0.000,B 0.000,C 90.000,E1 152.666} C_DIS
LIN {X 0.106,Y -523.333,Z 881.643,A 0.000,B 0.000,C 90.000,E1 151.769} C_DIS
LIN {X -0.131,Y -528.926,Z 881.638,A 0.000,B 0.000,C 90.000,E1 150.923} C_DIS
LIN {X -0.046,Y -534.294,Z 881.634,A 0.000,B 0.000,C 90.000,E1 150.049} C_DIS
LIN {X -0.310,Y -540.126,Z 881.628,A 0.000,B 0.000,C 90.000,E1 149.076} C_DIS
LIN {X -0.101,Y -544.890,Z 881.623,A 0.000,B 0.000,C 90.000,E1 148.201} C_DIS
LIN {X -0.042,Y -552.805,Z 881.615,A 0.000,B 0.000,C 90.000,E1 146.786} C_DIS
LIN {X 0.115,Y -559.291,Z 881.609,A 0.000,B 0.000,C 90.000,E1 145.515} C_DIS
LIN {X 0.174,Y -564.743,Z 881.602,A 0.000,B 0.000,C 90.000,E1 144.402} C_DIS
LIN {X -0.154,Y -570.257,Z 881.596,A 0.000,B 0.000,C 90.000,E1 143.336} C_DIS
LIN {X 0.006,Y -573.536,Z 881.592,A 0.000,B 0.000,C 90.000,E1 142.637} C_DIS
LIN {X -0.248,Y -580.676,Z 881.584,A 0.000,B 0.000,C 90.000,E1 141.170} C_DIS
LIN {X 0.087,Y -583.205,Z 881.581,A 0.000,B 0.000,C 90.000,E1 140.598} C_DIS
LIN {X 0.097,Y -589.252,Z 881.574,A 0.000,B 0.000,C 90.000,E1 139.256} C_DIS
LIN {X -0.081,Y -598.946,Z 881.562,A 0.000,B 0.000,C 90.000,E1 137.148} C_DIS
LIN {X 0.300,Y -606.952,Z 881.552,A 0.000,B 0.000,C 90.000,E1 135.405} C_DIS
LIN {X -0.102,Y -612.291,Z 881.546,A 0.000,B 0.000,C 90.000,E1 134.271} C_DIS
LIN {X 0.208,Y -619.120,Z 881.537,A 0.000,B 0.000,C 90.000,E1 132.690} C_DIS
LIN {X 0.058,Y -623.592,Z 881.532,A 0.000,B 0.000,C 90.000,E1 131.676} C_DIS
LIN {X 0.099,Y -626.817,Z 881.527,A 0.000,B 0.000,C 90.000,E1 130.906} C_DIS
LIN {X 0.115,Y -631.012,Z 881.522,A 0.000,B 0.000,C 90.000,E1 129.886} C_DIS
LIN {X -0.294,Y -635.021,Z 881.516,A 0.000,B 0.000,C 90.000,E1 128.910} C_DIS
LIN {X -0.377,Y -641.890,Z 881.506,A 0.000,B 0.000,C 90.000,E1 127.156} C_DIS
LIN {X -0.159,Y -645.654,Z 881.501,A 0.000,B 0.000,C 90.000,E1 126.137} C_DIS
LIN {X 0.256,Y -649.222,Z 881.495,A 0.000,B 0.000,C 90.000,E1 125.105} C_DIS
LIN {X -0.249,Y -651.713,Z 881.491,A 0.000,B 0.000,C 90.000,E1 124.405} C_DIS
LIN {X -0.199,Y -655.531,Z 881.484,A 0.000,B 0.000,C 90.000,E1 123.166} C_DIS
LIN {X -0.099,Y -657.664,Z 881.480,A 0.000,B 0.000,C 90.000,E1 122.418} C_DIS
LIN {X 0.138,Y -660.133,Z 881.475,A 0.000,B 0.000,C 90.000,E1 121.416} C_DIS
LIN {X -0.159,Y -662.138,Z 881.469,A 0.000,B 0.000,C 90.000,E1 120.463} C_DIS
LIN {X 0.106,Y -663.095,Z 881.466,A 0.000,B 0.000,C 90.000,E1 119.951} C_DIS
LIN {X -0.169,Y -664.704,Z 881.461,A 0.000,B 0.000,C 90.000,E1 118.999} C_DIS
LIN {X -0.023,Y -666.473,Z 881.454,A 0.000,B 0.000,C 90.000,E1 117.769} C_DIS
LIN {X -0.158,Y -667.575,Z 881.450,A 0.000,B 0.000,C 90.000,E1 117.052} C_DIS
LIN {X 0.014,Y -668.515,Z 881.446,A 0.000,B 0.000,C 90.000,E1 116.309} C_DIS
LIN {X 0.056,Y -669.492,Z 881.441,A 0.000,B 0.000,C 90.000,E1 115.335} C_DIS
LIN {X 0.262,Y -669.916,Z 881.437,A 0.000,B 0.000,C 90.000,E1 114.591} C_DIS
LIN {X -0.022,Y -670.056,Z 881.434,A 0.000,B 0.000,C 90.000,E1 114.131} C_DIS
LIN {X 0.031,Y -669.942,Z 881.431,A 0.000,B 0.000,C 90.000,E1 113.643} C_DIS
LIN {X 0.088,Y -669.236,Z 881.429,A 0.000,B 0.000,C 90.000,E1 113.153} C_DIS
LIN {X 0.248,Y -668.649,Z 881.427,A 0.000,B 0.000,C 90.000,E1 112.898} C_DIS
LIN {X 0.080,Y -665.561,Z 881.424,A 0.000,B 0.000,C 90.000,E1 112.333} C_DIS
LIN {X 0.153,Y -664.578,Z 881.423,A 0.000,B 0.000,C 90.000,E1 112.206} C_DIS
LIN {X 0.253,Y -659.525,Z 881.421,A 0.000,B 0.000,C 90.000,E1 111.716} C_DIS
LIN {X 0.357,Y -657.676,Z 881.420,A 0.000,B 0.000,C 90.000,E1 111.589} C_DIS
LIN {X -0.012,Y -648.026,Z 881.418,A 0.000,B 0.000,C 90.000,E1 111.227} C_DIS
LIN {X 0.079,Y -646.180,Z 881.418,A 0.000,B 0.000,C 90.000,E1 111.153} C_DIS
LIN {X 0.054,Y -635.180,Z 881.416,A 0.000,B 0.000,C 90.000,E1 110.865} C_DIS
LIN {X 0.095,Y -631.196,Z 881.415,A 0.000,B 0.000,C 90.000,E1 110.737} C_DIS
LIN {X 0.331,Y -627.147,Z 881.415,A 0.000,B 0.000,C 90.000,E1 110.610} C_DIS
LIN {X 0.009,Y -617.926,Z 881.413,A 0.000,B 0.000,C 90.000,E1 110.355} C_DIS
LIN {X 0.244,Y -611.977,Z 881.412,A 0.000,B 0.000,C 90.000,E1 110.120} C_DIS
LIN {X 0.080,Y -603.081,Z 881.410,A 0.000,B 0.000,C 90.000,E1 109.758} C_DIS
LIN {X -0.048,Y -588.076,Z 881.406,A 0.000,B 0.000,C 90.000,E1 109.033} C_DIS
LIN {X -0.120,Y -579.485,Z 881.404,A 0.000,B 0.000,C 90.000,E1 108.671} C_DIS
LIN {X 0.200,Y -565.551,Z 881.401,A 0.000,B 0.000,C 90.000,E1 108.181} C_DIS
LIN {X 0.005,Y -562.132,Z 881.400,A 0.000,B 0.000,C 90.000,E1 108.055} C_DIS
LIN {X -0.073,Y -559.386,Z 881.399,A 0.000,B 0.000,C 90.000,E1 107.873} C_DIS
LIN {X -0.117,Y -559.345,Z 881.399,A 0.000,B 0.000,C 90.000,E1 107.873} C_DIS
LIN {X -0.091,Y -557.931,Z 881.398,A 0.000,B 0.000,C 90.000,E1 107.583} C_DIS
LIN {X 0.275,Y -557.302,Z 881.395,A 0.000,B 0.000,C 90.000,E1 107.094} C_DIS
LIN {X 0.158,Y -558.316,Z 881.374,A 0.000,B 0.000,C 90.000,E1 103.355} C_DIS
LIN {X 0.070,Y -559.483,Z 881.364,A 0.000,B 0.000,C 90.000,E1 101.422} C_DIS
LIN {X -0.149,Y -560.658,Z 881.354,A 0.000,B 0.000,C 90.000,E1 99.782} C_DIS
LIN {X -0.134,Y -561.651,Z 881.347,A 0.000,B 0.000,C 90.000,E1 98.398} C_DIS
LIN {X -0.167,Y -562.339,Z 881.341,A 0.000,B 0.000,C 90.000,E1 97.296} C_DIS
LIN {X -0.115,Y -563.146,Z 881.333,A 0.000,B 0.000,C 90.000,E1 95.910} C_DIS
LIN {X -0.010,Y -563.931,Z 881.324,A 0.000,B 0.000,C 90.000,E1 94.245} C_DIS
LIN {X 0.011,Y -564.455,Z 881.316,A 0.000,B 0.000,C 90.000,E1 92.865} C_DIS
LIN {X 0.225,Y -565.083,Z 881.305,A 0.000,B 0.000,C 90.000,E1 90.917} C_DIS
LIN {X 0.220,Y -565.427,Z 881.298,A 0.000,B 0.000,C 90.000,E1 89.542} C_DIS
LIN {X -0.218,Y -565.741,Z 881.288,A 0.000,B 0.000,C 90.000,E1 87.936} C_DIS
LIN {X 0.023,Y -566.092,Z 881.278,A 0.000,B 0.000,C 90.000,E1 85.988} C_DIS
LIN {X 0.078,Y -566.296,Z 881.270,A 0.000,B 0.000,C 90.000,E1 84.609} C_DIS
LIN {X -0.105,Y -566.688,Z 881.259,A 0.000,B 0.000,C 90.000,E1 82.704} C_DIS
LIN {X -0.195,Y -567.204,Z 881.249,A 0.000,B 0.000,C 90.000,E1 80.792} C_DIS
LIN {X -0.175,Y -567.941,Z 881.238,A 0.000,B 0.000,C 90.000,E1 78.870} C_DIS
LIN {X 0.168,Y -568.576,Z 881.231,A 0.000,B 0.000,C 90.000,E1 77.465} C_DIS
LIN {X 0.141,Y -569.299,Z 881.221,A 0.000,B 0.000,C 90.000,E1 75.825} C_DIS
LIN {X 0.228,Y -569.846,Z 881.214,A 0.000,B 0.000,C 90.000,E1 74.448} C_DIS
LIN {X 0.172,Y -570.247,Z 881.206,A 0.000,B 0.000,C 90.000,E1 73.087} C_DIS
LIN {X 0.083,Y -570.637,Z 881.197,A 0.000,B 0.000,C 90.000,E1 71.456} C_DIS
LIN {X -0.002,Y -570.868,Z 881.188,A 0.000,B 0.000,C 90.000,E1 69.826} C_DIS
LIN {X -0.251,Y -571.051,Z 881.176,A 0.000,B 0.000,C 90.000,E1 67.667} C_DIS
LIN {X -0.056,Y -571.101,Z 881.168,A 0.000,B 0.000,C 90.000,E1 66.282} C_DIS
LIN {X -0.262,Y -571.070,Z 881.159,A 0.000,B 0.000,C 90.000,E1 64.665} C_DIS
LIN {X 0.177,Y -570.942,Z 881.152,A 0.000,B 0.000,C 90.000,E1 63.256} C_DIS
LIN {X -0.061,Y -570.591,Z 881.142,A 0.000,B 0.000,C 90.000,E1 61.641} C_DIS
LIN {X 0.138,Y -570.225,Z 881.135,A 0.000,B 0.000,C 90.000,E1 60.255} C_DIS
LIN {X -0.097,Y -569.873,Z 881.130,A 0.000,B 0.000,C 90.000,E1 59.459} C_DIS
LIN {X 0.082,Y -569.102,Z 881.123,A 0.000,B 0.000,C 90.000,E1 58.074} C_DIS
LIN {X 0.131,Y -568.523,Z 881.118,A 0.000,B 0.000,C 90.000,E1 57.248} C_DIS
LIN {X 0.177,Y -567.824,Z 881.114,A 0.000,B 0.000,C 90.000,E1 56.421} C_DIS
LIN {X 0.012,Y -566.743,Z 881.107,A 0.000,B 0.000,C 90.000,E1 55.341} C_DIS
LIN {X -0.315,Y -565.504,Z 881.101,A 0.000,B 0.000,C 90.000,E1 54.276} C_DIS
LIN {X 0.135,Y -563.965,Z 881.095,A 0.000,B 0.000,C 90.000,E1 53.130} C_DIS
LIN {X 0.011,Y -562.702,Z 881.091,A 0.000,B 0.000,C 90.000,E1 52.316} C_DIS
LIN {X 0.320,Y -561.320,Z 881.086,A 0.000,B 0.000,C 90.000,E1 51.457} C_DIS
LIN {X 0.173,Y -559.705,Z 881.081,A 0.000,B 0.000,C 90.000,E1 50.642} C_DIS
LIN {X -0.076,Y -558.552,Z 881.078,A 0.000,B 0.000,C 90.000,E1 50.114} C_DIS
LIN {X -0.251,Y -556.545,Z 881.074,A 0.000,B 0.000,C 90.000,E1 49.299} C_DIS
LIN {X -0.084,Y -554.134,Z 881.069,A 0.000,B 0.000,C 90.000,E1 48.447} C_DIS
LIN {X 0.059,Y -551.431,Z 881.065,A 0.000,B 0.000,C 90.000,E1 47.595} C_DIS
LIN {X -0.203,Y -548.432,Z 881.060,A 0.000,B 0.000,C 90.000,E1 46.782} C_DIS
LIN {X 0.248,Y -545.175,Z 881.055,A 0.000,B 0.000,C 90.000,E1 45.891} C_DIS
LIN {X 0.273,Y -542.806,Z 881.052,A 0.000,B 0.000,C 90.000,E1 45.324} C_DIS
LIN {X 0.087,Y -540.908,Z 881.050,A 0.000,B 0.000,C 90.000,E1 44.919} C_DIS
LIN {X 0.264,Y -537.391,Z 881.046,A 0.000,B 0.000,C 90.000,E1 44.190} C_DIS
LIN {X 0.228,Y -534.278,Z 881.043,A 0.000,B 0.000,C 90.000,E1 43.623} C_DIS
LIN {X -0.026,Y -530.086,Z 881.039,A 0.000,B 0.000,C 90.000,E1 42.933} C_DIS
LIN {X -0.277,Y -527.464,Z 881.036,A 0.000,B 0.000,C 90.000,E1 42.528} C_DIS
LIN {X 0.155,Y -522.759,Z 881.032,A 0.000,B 0.000,C 90.000,E1 41.757} C_DIS
LIN {X 0.254,Y -519.781,Z 881.030,A 0.000,B 0.000,C 90.000,E1 41.310} C_DIS
LIN {X 0.137,Y -512.208,Z 881.024,A 0.000,B 0.000,C 90.000,E1 40.297} C_DIS
LIN {X 0.081,Y -507.589,Z 881.021,A 0.000,B 0.000,C 90.000,E1 39.725} C_DIS
LIN {X 0.203,Y -502.512,Z 881.018,A 0.000,B 0.000,C 90.000,E1 39.116} C_DIS
LIN {X -0.085,Y -498.576,Z 881.015,A 0.000,B 0.000,C 90.000,E1 38.705} C_DIS
LIN {X 0.227,Y -490.307,Z 881.010,A 0.000,B 0.000,C 90.000,E1 37.810} C_DIS
LIN {X -0.031,Y -484.616,Z 881.007,A 0.000,B 0.000,C 90.000,E1 37.282} C_DIS
LIN {X 0.159,Y -477.138,Z 881.003,A 0.000,B 0.000,C 90.000,E1 36.583} C_DIS
LIN {X 0.174,Y -469.647,Z 881.000,A 0.000,B 0.000,C 90.000,E1 35.931} C_DIS
LIN {X -0.020,Y -462.061,Z 880.996,A 0.000,B 0.000,C 90.000,E1 35.311} C_DIS
LIN {X 0.210,Y -451.180,Z 880.991,A 0.000,B 0.000,C 90.000,E1 34.405} C_DIS
LIN {X -0.206,Y -434.043,Z 880.984,A 0.000,B 0.000,C 90.000,E1 33.086} C_DIS
LIN {X 0.178,Y -420.230,Z 880.977,A 0.000,B 0.000,C 90.000,E1 31.878} C_DIS
LIN {X 0.010,Y -406.753,Z 880.970,A 0.000,B 0.000,C 90.000,E1 30.669} C_DIS
LIN {X -0.037,Y -399.723,Z 880.966,A 0.000,B 0.000,C 90.000,E1 29.951} C_DIS
LIN {X 0.063,Y -396.819,Z 880.965,A 0.000,B 0.000,C 90.000,E1 29.617} C_DIS
LIN {X 0.083,Y -393.783,Z 880.962,A 0.000,B 0.000,C 90.000,E1 29.205} C_DIS
LIN {X 0.012,Y -393.260,Z 880.962,A 0.000,B 0.000,C 90.000,E1 29.127} C_DIS
LIN {X 0.184,Y -391.068,Z 880.959,A 0.000,B 0.000,C 90.000,E1 28.615} C_DIS
LIN {X 0.076,Y -390.233,Z 880.957,A 0.000,B 0.000,C 90.000,E1 28.231} C_DIS
LIN {X 0.081,Y -389.756,Z 880.956,A 0.000,B 0.000,C 90.000,E1 28.052} C_DIS
LIN {X -0.174,Y -389.173,Z 880.952,A 0.000,B 0.000,C 90.000,E1 27.385} C_DIS
LIN {X 0.200,Y -389.187,Z 880.948,A 0.000,B 0.000,C 90.000,E1 26.616} C_DIS
LIN {X -0.060,Y -392.598,Z 880.922,A 0.000,B 0.000,C 90.000,E1 22.025} C_DIS
LIN {X 0.029,Y -394.759,Z 880.911,A 0.000,B 0.000,C 90.000,E1 19.885} C_DIS
LIN {X 0.113,Y -397.548,Z 880.897,A 0.000,B 0.000,C 90.000,E1 17.402} C_DIS
LIN {X 0.035,Y -400.561,Z 880.883,A 0.000,B 0.000,C 90.000,E1 14.954} C_DIS
LIN {X -0.149,Y -402.918,Z 880.873,A 0.000,B 0.000,C 90.000,E1 13.231} C_DIS
LIN {X -0.066,Y -406.427,Z 880.860,A 0.000,B 0.000,C 90.000,E1 10.782} C_DIS
LIN {X 0.063,Y -410.281,Z 880.846,A 0.000,B 0.000,C 90.000,E1 8.341} C_DIS
LIN {X -0.183,Y -415.090,Z 880.831,A 0.000,B 0.000,C 90.000,E1 5.625} C_DIS
LIN {X 0.000,Y -419.654,Z 880.818,A 0.000,B 0.000,C 90.000,E1 3.212} C_DIS
LIN {X -0.083,Y -425.520,Z 880.803,A 0.000,B 0.000,C 90.000,E1 0.516} C_DIS
LIN {X -0.076,Y -429.604,Z 880.793,A 0.000,B 0.000,C 90.000,E1 358.797} C_DIS
LIN {X -0.015,Y -434.589,Z 880.782,A 0.000,B 0.000,C 90.000,E1 356.788} C_DIS
LIN {X -0.153,Y -437.191,Z 880.777,A 0.000,B 0.000,C 90.000,E1 355.812} C_DIS
LIN {X 0.073,Y -439.283,Z 880.773,A 0.000,B 0.000,C 90.000,E1 355.122} C_DIS
LIN {X -0.213,Y -441.550,Z 880.770,A 0.000,B 0.000,C 90.000,E1 354.666} C_DIS
LIN {X -0.119,Y -442.439,Z 880.769,A 0.000,B 0.000,C 90.000,E1 354.489} C_DIS
LIN {X 0.102,Y -444.720,Z 880.768,A 0.000,B 0.000,C 90.000,E1 354.147} C_DIS
LIN {X 0.033,Y -447.556,Z 880.766,A 0.000,B 0.000,C 90.000,E1 353.913} C_DIS
LIN {X -0.120,Y -450.385,Z 880.765,A 0.000,B 0.000,C 90.000,E1 353.742} C_DIS
LIN {X -0.123,Y -456.148,Z 880.764,A 0.000,B 0.000,C 90.000,E1 353.451} C_DIS
LIN {X 0.121,Y -466.110,Z 880.761,A 0.000,B 0.000,C 90.000,E1 352.996} C_DIS
LIN {X 0.092,Y -476.085,Z 880.759,A 0.000,B 0.000,C 90.000,E1 352.534} C_DIS
LIN {X 0.191,Y -482.414,Z 880.757,A 0.000,B 0.000,C 90.000,E1 352.186} C_DIS
LIN {X 0.041,Y -489.082,Z 880.755,A 0.000,B 0.000,C 90.000,E1 351.837} C_DIS
LIN {X -0.154,Y -500.429,Z 880.751,A 0.000,B 0.000,C 90.000,E1 351.197} C_DIS
LIN {X 0.156,Y -509.942,Z 880.748,A 0.000,B 0.000,C 90.000,E1 350.566} C_DIS
LIN {X 0.230,Y -517.748,Z 880.745,A 0.000,B 0.000,C 90.000,E1 350.038} C_DIS
LIN {X 0.120,Y -525.429,Z 880.742,A 0.000,B 0.000,C 90.000,E1 349.511} C_DIS
LIN {X -0.221,Y -531.488,Z 880.739,A 0.000,B 0.000,C 90.000,E1 349.106} C_DIS
LIN {X -0.207,Y -538.761,Z 880.736,A 0.000,B 0.000,C 90.000,E1 348.522} C_DIS
LIN {X 0.149,Y -545.675,Z 880.733,A 0.000,B 0.000,C 90.000,E1 347.881} C_DIS
LIN {X 0.207,Y -553.669,Z 880.729,A 0.000,B 0.000,C 90.000,E1 347.117} C_DIS
LIN {X -0.064,Y -557.569,Z 880.726,A 0.000,B 0.000,C 90.000,E1 346.756} C_DIS
LIN {X -0.163,Y -562.650,Z 880.723,A 0.000,B 0.000,C 90.000,E1 346.228} C_DIS
LIN {X 0.168,Y -567.521,Z 880.720,A 0.000,B 0.000,C 90.000,E1 345.644} C_DIS
LIN {X 0.109,Y -572.107,Z 880.717,A 0.000,B 0.000,C 90.000,E1 345.102} C_DIS
LIN {X 0.133,Y -578.520,Z 880.713,A 0.000,B 0.000,C 90.000,E1 344.283} C_DIS
LIN {X 0.069,Y -583.519,Z 880.709,A 0.000,B 0.000,C 90.000,E1 343.614} C_DIS
LIN {X -0.192,Y -589.024,Z 880.705,A 0.000,B 0.000,C 90.000,E1 342.834} C_DIS
LIN {X 0.229,Y -593.302,Z 880.701,A 0.000,B 0.000,C 90.000,E1 342.127} C_DIS
LIN {X 0.058,Y -598.152,Z 880.696,A 0.000,B 0.000,C 90.000,E1 341.348} C_DIS
LIN {X 0.044,Y -604.121,Z 880.691,A 0.000,B 0.000,C 90.000,E1 340.296} C_DIS
LIN {X -0.023,Y -608.300,Z 880.686,A 0.000,B 0.000,C 90.000,E1 339.518} C_DIS
LIN {X 0.115,Y -613.725,Z 880.680,A 0.000,B 0.000,C 90.000,E1 338.465} C_DIS
LIN {X 0.346,Y -618.232,Z 880.675,A 0.000,B 0.000,C 90.000,E1 337.539} C_DIS
LIN {X 0.054,Y -623.640,Z 880.669,A 0.000,B 0.000,C 90.000,E1 336.410} C_DIS
LIN {X -0.173,Y -628.148,Z 880.663,A 0.000,B 0.000,C 90.000,E1 335.409} C_DIS
LIN {X -0.351,Y -632.290,Z 880.658,A 0.000,B 0.000,C 90.000,E1 334.409} C_DIS
LIN {X -0.158,Y -637.099,Z 880.651,A 0.000,B 0.000,C 90.000,E1 333.127} C_DIS
LIN {X 0.054,Y -640.669,Z 880.645,A 0.000,B 0.000,C 90.000,E1 332.103} C_DIS
LIN {X 0.126,Y -644.768,Z 880.638,A 0.000,B 0.000,C 90.000,E1 330.845} C_DIS
LIN {X 0.358,Y -649.293,Z 880.630,A 0.000,B 0.000,C 90.000,E1 329.331} C_DIS
LIN {X 0.112,Y -653.449,Z 880.622,A 0.000,B 0.000,C 90.000,E1 327.867} C_DIS
LIN {X -0.269,Y -655.949,Z 880.616,A 0.000,B 0.000,C 90.000,E1 326.914} C_DIS
LIN {X 0.294,Y -658.204,Z 880.611,A 0.000,B 0.000,C 90.000,E1 325.881} C_DIS
LIN {X -0.098,Y -660.561,Z 880.604,A 0.000,B 0.000,C 90.000,E1 324.689} C_DIS
LIN {X -0.062,Y -662.511,Z 880.597,A 0.000,B 0.000,C 90.000,E1 323.463} C_DIS
LIN {X -0.392,Y -664.241,Z 880.590,A 0.000,B 0.000,C 90.000,E1 322.271} C_DIS
LIN {X -0.322,Y -665.860,Z 880.582,A 0.000,B 0.000,C 90.000,E1 320.803} C_DIS
LIN {X 0.212,Y -667.197,Z 880.575,A 0.000,B 0.000,C 90.000,E1 319.542} C_DIS
LIN {X 0.263,Y -668.771,Z 880.567,A 0.000,B 0.000,C 90.000,E1 318.081} C_DIS
LIN {X 0.353,Y -670.595,Z 880.558,A 0.000,B 0.000,C 90.000,E1 316.377} C_DIS
LIN {X -0.017,Y -672.439,Z 880.548,A 0.000,B 0.000,C 90.000,E1 314.717} C_DIS
LIN {X 0.100,Y -673.604,Z 880.542,A 0.000,B 0.000,C 90.000,E1 313.500} C_DIS
LIN {X 0.216,Y -674.843,Z 880.535,A 0.000,B 0.000,C 90.000,E1 312.285} C_DIS
LIN {X -0.032,Y -676.141,Z 880.527,A 0.000,B 0.000,C 90.000,E1 310.862} C_DIS
LIN {X -0.224,Y -677.558,Z 880.518,A 0.000,B 0.000,C 90.000,E1 309.197} C_DIS
LIN {X 0.091,Y -678.506,Z 880.511,A 0.000,B 0.000,C 90.000,E1 307.971} C_DIS
LIN {X -0.118,Y -679.436,Z 880.504,A 0.000,B 0.000,C 90.000,E1 306.790} C_DIS
LIN {X -0.179,Y -680.314,Z 880.498,A 0.000,B 0.000,C 90.000,E1 305.598} C_DIS
LIN {X -0.049,Y -681.272,Z 880.488,A 0.000,B 0.000,C 90.000,E1 303.913} C_DIS
LIN {X 0.113,Y -682.074,Z 880.482,A 0.000,B 0.000,C 90.000,E1 302.704} C_DIS
LIN {X -0.290,Y -683.749,Z 880.470,A 0.000,B 0.000,C 90.000,E1 300.590} C_DIS
LIN {X -0.167,Y -685.623,Z 880.458,A 0.000,B 0.000,C 90.000,E1 298.437} C_DIS
LIN {X -0.215,Y -687.690,Z 880.447,A 0.000,B 0.000,C 90.000,E1 296.539} C_DIS
LIN {X 0.234,Y -689.360,Z 880.440,A 0.000,B 0.000,C 90.000,E1 295.079} C_DIS
LIN {X -0.037,Y -690.192,Z 880.434,A 0.000,B 0.000,C 90.000,E1 294.155} C_DIS
LIN {X -0.245,Y -690.582,Z 880.430,A 0.000,B 0.000,C 90.000,E1 293.462} C_DIS
LIN {X 0.220,Y -690.257,Z 880.428,A 0.000,B 0.000,C 90.000,E1 292.950} C_DIS
LIN {X 0.183,Y -690.011,Z 880.426,A 0.000,B 0.000,C 90.000,E1 292.717} C_DIS
LIN {X -0.258,Y -688.428,Z 880.424,A 0.000,B 0.000,C 90.000,E1 292.280} C_DIS
LIN {X -0.034,Y -687.441,Z 880.422,A 0.000,B 0.000,C 90.000,E1 292.025} C_DIS
LIN {X 0.076,Y -686.565,Z 880.422,A 0.000,B 0.000,C 90.000,E1 291.897} C_DIS
LIN {X 0.078,Y -683.916,Z 880.420,A 0.000,B 0.000,C 90.000,E1 291.663} C_DIS
LIN {X -0.033,Y -679.453,Z 880.419,A 0.000,B 0.000,C 90.000,E1 291.354} C_DIS
LIN {X 0.317,Y -677.334,Z 880.418,A 0.000,B 0.000,C 90.000,E1 291.227} C_DIS
LIN {X 0.343,Y -668.967,Z 880.417,A 0.000,B 0.000,C 90.000,E1 290.972} C_DIS
LIN {X 0.339,Y -662.009,Z 880.416,A 0.000,B 0.000,C 90.000,E1 290.791} C_DIS
LIN {X -0.256,Y -659.261,Z 880.415,A 0.000,B 0.000,C 90.000,E1 290.737} C_DIS
LIN {X -0.269,Y -655.225,Z 880.414,A 0.000,B 0.000,C 90.000,E1 290.556} C_DIS
LIN {X -0.094,Y -655.158,Z 880.414,A 0.000,B 0.000,C 90.000,E1 290.536} C_DIS
LIN {X 0.111,Y -653.927,Z 880.413,A 0.000,B 0.000,C 90.000,E1 290.375} C_DIS
LIN {X 0.067,Y -653.916,Z 880.413,A 0.000,B 0.000,C 90.000,E1 290.375} C_DIS
LIN {X 0.252,Y -653.758,Z 880.412,A 0.000,B 0.000,C 90.000,E1 290.174} C_DIS
LIN {X 0.208,Y -654.163,Z 880.411,A 0.000,B 0.000,C 90.000,E1 289.993} C_DIS
LIN {X 0.075,Y -654.865,Z 880.410,A 0.000,B 0.000,C 90.000,E1 289.758} C_DIS
LIN {X 0.408,Y -658.646,Z 880.406,A 0.000,B 0.000,C 90.000,E1 288.960} C_DIS
LIN {X 0.253,Y -664.509,Z 880.399,A 0.000,B 0.000,C 90.000,E1 287.873} C_DIS
LIN {X -0.016,Y -667.960,Z 880.395,A 0.000,B 0.000,C 90.000,E1 287.166} C_DIS
LIN {X -0.054,Y -670.929,Z 880.391,A 0.000,B 0.000,C 90.000,E1 286.441} C_DIS
LIN {X -0.190,Y -672.627,Z 880.389,A 0.000,B 0.000,C 90.000,E1 285.969} C_DIS
LIN {X -0.192,Y -674.663,Z 880.385,A 0.000,B 0.000,C 90.000,E1 285.245} C_DIS
LIN {X -0.303,Y -675.778,Z 880.382,A 0.000,B 0.000,C 90.000,E1 284.773} C_DIS
LIN {X 0.202,Y -677.140,Z 880.378,A 0.000,B 0.000,C 90.000,E1 284.008} C_DIS
LIN {X 0.067,Y -678.192,Z 880.374,A 0.000,B 0.000,C 90.000,E1 283.300} C_DIS
LIN {X -0.018,Y -678.775,Z 880.371,A 0.000,B 0.000,C 90.000,E1 282.827} C_DIS
LIN {X -0.144,Y -679.394,Z 880.367,A 0.000,B 0.000,C 90.000,E1 282.119} C_DIS
LIN {X -0.366,Y -679.619,Z 880.365,A 0.000,B 0.000,C 90.000,E1 281.658} C_DIS
LIN {X 0.261,Y -679.703,Z 880.363,A 0.000,B 0.000,C 90.000,E1 281.366} C_DIS
LIN {X 0.136,Y -679.377,Z 880.359,A 0.000,B 0.000,C 90.000,E1 280.658} C_DIS
LIN {X -0.075,Y -678.932,Z 880.357,A 0.000,B 0.000,C 90.000,E1 280.197} C_DIS
LIN {X -0.168,Y -678.197,Z 880.354,A 0.000,B 0.000,C 90.000,E1 279.726} C_DIS
LIN {X 0.231,Y -676.470,Z 880.350,A 0.000,B 0.000,C 90.000,E1 278.973} C_DIS
LIN {X 0.011,Y -674.979,Z 880.347,A 0.000,B 0.000,C 90.000,E1 278.511} C_DIS
LIN {X -0.217,Y -673.202,Z 880.345,A 0.000,B 0.000,C 90.000,E1 278.049} C_DIS
LIN {X 0.214,Y -671.102,Z 880.342,A 0.000,B 0.000,C 90.000,E1 277.530} C_DIS
LIN {X -0.037,Y -668.097,Z 880.339,A 0.000,B 0.000,C 90.000,E1 276.947} C_DIS
LIN {X 0.264,Y -664.591,Z 880.335,A 0.000,B 0.000,C 90.000,E1 276.315} C_DIS
LIN {X -0.031,Y -661.451,Z 880.333,A 0.000,B 0.000,C 90.000,E1 275.853} C_DIS
LIN {X 0.311,Y -657.857,Z 880.330,A 0.000,B 0.000,C 90.000,E1 275.334} C_DIS
LIN {X -0.084,Y -653.723,Z 880.327,A 0.000,B 0.000,C 90.000,E1 274.878} C_DIS
LIN {X 0.112,Y -647.861,Z 880.324,A 0.000,B 0.000,C 90.000,E1 274.245} C_DIS
LIN {X -0.124,Y -642.765,Z 880.321,A 0.000,B 0.000,C 90.000,E1 273.784} C_DIS
LIN {X -0.226,Y -637.463,Z 880.318,A 0.000,B 0.000,C 90.000,E1 273.326} C_DIS
LIN {X -0.048,Y -630.463,Z 880.315,A 0.000,B 0.000,C 90.000,E1 272.751} C_DIS
LIN {X -0.255,Y -624.484,Z 880.313,A 0.000,B 0.000,C 90.000,E1 272.350} C_DIS
LIN {X 0.067,Y -616.556,Z 880.310,A 0.000,B 0.000,C 90.000,E1 271.835} C_DIS
LIN {X -0.036,Y -609.945,Z 880.308,A 0.000,B 0.000,C 90.000,E1 271.489} C_DIS
LIN {X 0.200,Y -603.095,Z 880.307,A 0.000,B 0.000,C 90.000,E1 271.146} C_DIS
LIN {X 0.282,Y -597.900,Z 880.305,A 0.000,B 0.000,C 90.000,E1 270.917} C_DIS
LIN {X -0.119,Y -590.569,Z 880.304,A 0.000,B 0.000,C 90.000,E1 270.688} C_DIS
LIN {X -0.160,Y -584.595,Z 880.303,A 0.000,B 0.000,C 90.000,E1 270.516} C_DIS
LIN {X 0.248,Y -577.180,Z 880.302,A 0.000,B 0.000,C 90.000,E1 270.286} C_DIS
LIN {X 0.242,Y -571.326,Z 880.301,A 0.000,B 0.000,C 90.000,E1 270.172} C_DIS
LIN {X -0.125,Y -562.849,Z 880.301,A 0.000,B 0.000,C 90.000,E1 270.115} C_DIS
LIN {X -0.107,Y -554.527,Z 880.300,A 0.000,B 0.000,C 90.000,E1 270.057} C_DIS
LIN {X 0.122,Y -551.943,Z 880.300,A 0.000,B 0.000,C 90.000,E1 270.000} C_DIS
LIN {X -0.011,Y -549.252,Z 880.300,A 0.000,B 0.000,C 90.000,E1 269.943} C_DIS
LIN {X -0.039,Y -549.197,Z 880.300,A 0.000,B 0.000,C 90.000,E1 269.943} C_DIS
LIN {X 0.272,Y -546.994,Z 880.298,A 0.000,B 0.000,C 90.000,E1 269.656} C_DIS
LIN {X -0.100,Y -546.157,Z 880.297,A 0.000,B 0.000,C 90.000,E1 269.484} C_DIS
LIN {X -0.080,Y -545.241,Z 880.295,A 0.000,B 0.000,C 90.000,E1 269.026} C_DIS
LIN {X -0.091,Y -541.727,Z 880.273,A 0.000,B 0.000,C 90.000,E1 265.065} C_DIS
LIN {X 0.076,Y -540.805,Z 880.265,A 0.000,B 0.000,C 90.000,E1 263.628} C_DIS
LIN {X 0.283,Y -539.966,Z 880.258,A 0.000,B 0.000,C 90.000,E1 262.470} C_DIS
LIN {X -0.132,Y -538.906,Z 880.252,A 0.000,B 0.000,C 90.000,E1 261.376} C_DIS
LIN {X 0.170,Y -537.141,Z 880.243,A 0.000,B 0.000,C 90.000,E1 259.634} C_DIS
LIN {X 0.005,Y -535.374,Z 880.233,A 0.000,B 0.000,C 90.000,E1 257.937} C_DIS
LIN {X -0.301,Y -534.043,Z 880.227,A 0.000,B 0.000,C 90.000,E1 256.825} C_DIS
LIN {X 0.230,Y -531.889,Z 880.217,A 0.000,B 0.000,C 90.000,E1 255.046} C_DIS
LIN {X 0.204,Y -529.771,Z 880.208,A 0.000,B 0.000,C 90.000,E1 253.323} C_DIS
LIN {X -0.224,Y -527.744,Z 880.198,A 0.000,B 0.000,C 90.000,E1 251.638} C_DIS
LIN {X -0.028,Y -525.480,Z 880.188,A 0.000,B 0.000,C 90.000,E1 249.880} C_DIS
LIN {X 0.130,Y -523.563,Z 880.180,A 0.000,B 0.000,C 90.000,E1 248.411} C_DIS
LIN {X 0.288,Y -521.830,Z 880.174,A 0.000,B 0.000,C 90.000,E1 247.230} C_DIS
LIN {X 0.091,Y -519.641,Z 880.166,A 0.000,B 0.000,C 90.000,E1 245.793} C_DIS
LIN {X 0.206,Y -516.939,Z 880.156,A 0.000,B 0.000,C 90.000,E1 244.024} C_DIS
LIN {X 0.014,Y -515.027,Z 880.149,A 0.000,B 0.000,C 90.000,E1 242.871} C_DIS
LIN {X -0.214,Y -511.929,Z 880.140,A 0.000,B 0.000,C 90.000,E1 241.129} C_DIS
LIN {X -0.013,Y -508.877,Z 880.130,A 0.000,B 0.000,C 90.000,E1 239.331} C_DIS
LIN {X 0.173,Y -506.728,Z 880.123,A 0.000,B 0.000,C 90.000,E1 238.122} C_DIS
LIN {X 0.009,Y -505.056,Z 880.118,A 0.000,B 0.000,C 90.000,E1 237.248} C_DIS
LIN {X -0.292,Y -502.654,Z 880.111,A 0.000,B 0.000,C 90.000,E1 236.087} C_DIS
LIN {X -0.225,Y -500.729,Z 880.106,A 0.000,B 0.000,C 90.000,E1 235.182} C_DIS
LIN {X 0.131,Y -496.471,Z 880.096,A 0.000,B 0.000,C 90.000,E1 233.336} C_DIS
LIN {X 0.138,Y -493.019,Z 880.088,A 0.000,B 0.000,C 90.000,E1 231.823} C_DIS
LIN {X -0.151,Y -490.153,Z 880.081,A 0.000,B 0.000,C 90.000,E1 230.642} C_DIS
LIN {X 0.036,Y -486.695,Z 880.073,A 0.000,B 0.000,C 90.000,E1 229.094} C_DIS
LIN {X -0.036,Y -483.917,Z 880.066,A 0.000,B 0.000,C 90.000,E1 227.877} C_DIS
LIN {X -0.247,Y -479.918,Z 880.056,A 0.000,B 0.000,C 90.000,E1 226.053} C_DIS
LIN {X -0.209,Y -475.747,Z 880.045,A 0.000,B 0.000,C 90.000,E1 224.190} C_DIS
LIN {X -0.024,Y -472.302,Z 880.037,A 0.000,B 0.000,C 90.000,E1 222.609} C_DIS
LIN {X 0.203,Y -468.091,Z 880.026,A 0.000,B 0.000,C 90.000,E1 220.701} C_DIS
LIN {X -0.021,Y -464.662,Z 880.018,A 0.000,B 0.000,C 90.000,E1 219.152} C_DIS
LIN {X -0.024,Y -461.339,Z 880.009,A 0.000,B 0.000,C 90.000,E1 217.569} C_DIS
LIN {X 0.075,Y -457.994,Z 880.000,A 0.000,B 0.000,C 90.000,E1 215.964} C_DIS
LIN {X 0.103,Y -453.959,Z 879.989,A 0.000,B 0.000,C 90.000,E1 214.040} C_DIS
LIN {X 0.101,Y -451.160,Z 879.982,A 0.000,B 0.000,C 90.000,E1 212.752} C_DIS
LIN {X 0.059,Y -448.487,Z 879.975,A 0.000,B 0.000,C 90.000,E1 211.465} C_DIS
LIN {X -0.060,Y -443.624,Z 879.962,A 0.000,B 0.000,C 90.000,E1 209.205} C_DIS
LIN {X -0.020,Y -439.959,Z 879.953,A 0.000,B 0.000,C 90.000,E1 207.564} C_DIS
LIN {X -0.042,Y -435.655,Z 879.942,A 0.000,B 0.000,C 90.000,E1 205.591} C_DIS
LIN {X 0.057,Y -431.502,Z 879.931,A 0.000,B 0.000,C 90.000,E1 203.590} C_DIS
LIN {X 0.055,Y -427.276,Z 879.920,A 0.000,B 0.000,C 90.000,E1 201.589} C_DIS
LIN {X -0.156,Y -423.942,Z 879.911,A 0.000,B 0.000,C 90.000,E1 199.939} C_DIS
LIN {X -0.217,Y -419.177,Z 879.898,A 0.000,B 0.000,C 90.000,E1 197.583} C_DIS
LIN {X -0.080,Y -416.421,Z 879.890,A 0.000,B 0.000,C 90.000,E1 196.205} C_DIS
LIN {X 0.175,Y -412.245,Z 879.879,A 0.000,B 0.000,C 90.000,E1 194.120} C_DIS
LIN {X -0.039,Y -410.334,Z 879.873,A 0.000,B 0.000,C 90.000,E1 193.119} C_DIS
LIN {X -0.219,Y -406.269,Z 879.861,A 0.000,B 0.000,C 90.000,E1 191.074} C_DIS
LIN {X -0.102,Y -403.599,Z 879.854,A 0.000,B 0.000,C 90.000,E1 189.670} C_DIS
LIN {X -0.181,Y -399.310,Z 879.842,A 0.000,B 0.000,C 90.000,E1 187.587} C_DIS
LIN {X -0.044,Y -394.664,Z 879.828,A 0.000,B 0.000,C 90.000,E1 185.106} C_DIS
LIN {X -0.193,Y -390.071,Z 879.813,A 0.000,B 0.000,C 90.000,E1 182.293} C_DIS
LIN {X -0.032,Y -386.433,Z 879.799,A 0.000,B 0.000,C 90.000,E1 179.771} C_DIS
LIN {X -0.050,Y -384.343,Z 879.791,A 0.000,B 0.000,C 90.000,E1 178.339} C_DIS
LIN {X 0.192,Y -381.622,Z 879.781,A 0.000,B 0.000,C 90.000,E1 176.502} C_DIS
LIN {X -0.103,Y -378.409,Z 879.769,A 0.000,B 0.000,C 90.000,E1 174.375} C_DIS
LIN {X -0.064,Y -375.707,Z 879.757,A 0.000,B 0.000,C 90.000,E1 172.186} C_DIS
LIN {X -0.133,Y -374.507,Z 879.748,A 0.000,B 0.000,C 90.000,E1 170.735} C_DIS
LIN {X -0.152,Y -374.010,Z 879.740,A 0.000,B 0.000,C 90.000,E1 169.275} C_DIS
LIN {X -0.016,Y -374.158,Z 879.736,A 0.000,B 0.000,C 90.000,E1 168.522} C_DIS
LIN {X -0.048,Y -374.528,Z 879.734,A 0.000,B 0.000,C 90.000,E1 168.173} C_DIS
LIN {X -0.185,Y -374.919,Z 879.731,A 0.000,B 0.000,C 90.000,E1 167.645} C_DIS
LIN {X 0.048,Y -375.730,Z 879.728,A 0.000,B 0.000,C 90.000,E1 167.061} C_DIS
LIN {X 0.017,Y -376.120,Z 879.726,A 0.000,B 0.000,C 90.000,E1 166.700} C_DIS
LIN {X 0.045,Y -377.610,Z 879.723,A 0.000,B 0.000,C 90.000,E1 166.117} C_DIS
LIN {X 0.031,Y -379.552,Z 879.720,A 0.000,B 0.000,C 90.000,E1 165.574} C_DIS
LIN {X -0.078,Y -383.176,Z 879.716,A 0.000,B 0.000,C 90.000,E1 164.866} C_DIS
LIN {X 0.170,Y -389.229,Z 879.712,A 0.000,B 0.000,C 90.000,E1 164.157} C_DIS
LIN {X 0.141,Y -395.717,Z 879.710,A 0.000,B 0.000,C 90.000,E1 163.685} C_DIS
LIN {X 0.217,Y -416.119,Z 879.704,A 0.000,B 0.000,C 90.000,E1 162.598} C_DIS
LIN {X -0.014,Y -420.816,Z 879.702,A 0.000,B 0.000,C 90.000,E1 162.362} C_DIS
LIN {X -0.176,Y -424.194,Z 879.701,A 0.000,B 0.000,C 90.000,E1 162.181} C_DIS
LIN {X -0.212,Y -430.425,Z 879.699,A 0.000,B 0.000,C 90.000,E1 161.764} C_DIS
LIN {X 0.093,Y -438.341,Z 879.695,A 0.000,B 0.000,C 90.000,E1 161.148} C_DIS
LIN {X -0.016,Y -444.575,Z 879.693,A 0.000,B 0.000,C 90.000,E1 160.678} C_DIS
LIN {X -0.105,Y -452.217,Z 879.689,A 0.000,B 0.000,C 90.000,E1 160.061} C_DIS
LIN {X 0.217,Y -461.004,Z 879.685,A 0.000,B 0.000,C 90.000,E1 159.209} C_DIS
LIN {X -0.053,Y -467.857,Z 879.681,A 0.000,B 0.000,C 90.000,E1 158.539} C_DIS
LIN {X 0.199,Y -474.732,Z 879.677,A 0.000,B 0.000,C 90.000,E1 157.794} C_DIS
LIN {X -0.170,Y -483.965,Z 879.671,A 0.000,B 0.000,C 90.000,E1 156.794} C_DIS
LIN {X 0.095,Y -487.580,Z 879.668,A 0.000,B 0.000,C 90.000,E1 156.305} C_DIS
LIN {X 0.030,Y -489.816,Z 879.667,A 0.000,B 0.000,C 90.000,E1 156.049} C_DIS
LIN {X 0.039,Y -495.736,Z 879.663,A 0.000,B 0.000,C 90.000,E1 155.305} C_DIS
LIN {X -0.043,Y -502.506,Z 879.658,A 0.000,B 0.000,C 90.000,E1 154.409} C_DIS
LIN {X 0.041,Y -511.068,Z 879.651,A 0.000,B 0.000,C 90.000,E1 153.204} C_DIS
LIN {X -0.155,Y -516.088,Z 879.647,A 0.000,B 0.000,C 90.000,E1 152.487} C_DIS
LIN {X -0.089,Y -524.008,Z 879.641,A 0.000,B 0.000,C 90.000,E1 151.307} C_DIS
LIN {X -0.009,Y -527.740,Z 879.637,A 0.000,B 0.000,C 90.000,E1 150.717} C_DIS
LIN {X -0.051,Y -532.344,Z 879.633,A 0.000,B 0.000,C 90.000,E1 149.999} C_DIS
LIN {X -0.210,Y -539.104,Z 879.627,A 0.000,B 0.000,C 90.000,E1 148.869} C_DIS
LIN {X 0.012,Y -545.427,Z 879.621,A 0.000,B 0.000,C 90.000,E1 147.709} C_DIS
LIN {X 0.158,Y -551.011,Z 879.615,A 0.000,B 0.000,C 90.000,E1 146.707} C_DIS
LIN {X -0.095,Y -556.181,Z 879.610,A 0.000,B 0.000,C 90.000,E1 145.754} C_DIS
LIN {X 0.025,Y -561.047,Z 879.604,A 0.000,B 0.000,C 90.000,E1 144.769} C_DIS
LIN {X 0.111,Y -569.994,Z 879.594,A 0.000,B 0.000,C 90.000,E1 142.970} C_DIS
LIN {X -0.291,Y -573.972,Z 879.590,A 0.000,B 0.000,C 90.000,E1 142.190} C_DIS
LIN {X -0.087,Y -581.106,Z 879.582,A 0.000,B 0.000,C 90.000,E1 140.678} C_DIS
LIN {X 0.351,Y -584.898,Z 879.577,A 0.000,B 0.000,C 90.000,E1 139.828} C_DIS
LIN {X 0.112,Y -594.581,Z 879.565,A 0.000,B 0.000,C 90.000,E1 137.715} C_DIS
LIN {X 0.057,Y -599.541,Z 879.559,A 0.000,B 0.000,C 90.000,E1 136.662} C_DIS
LIN {X 0.315,Y -605.798,Z 879.552,A 0.000,B 0.000,C 90.000,E1 135.324} C_DIS
LIN {X -0.018,Y -610.529,Z 879.546,A 0.000,B 0.000,C 90.000,E1 134.312} C_DIS
LIN {X -0.175,Y -617.412,Z 879.538,A 0.000,B 0.000,C 90.000,E1 132.771} C_DIS
LIN {X -0.349,Y -621.936,Z 879.532,A 0.000,B 0.000,C 90.000,E1 131.757} C_DIS
LIN {X 0.145,Y -625.173,Z 879.528,A 0.000,B 0.000,C 90.000,E1 130.943} C_DIS
LIN {X 0.069,Y -629.398,Z 879.522,A 0.000,B 0.000,C 90.000,E1 129.930} C_DIS
LIN {X 0.125,Y -633.384,Z 879.516,A 0.000,B 0.000,C 90.000,E1 128.910} C_DIS
LIN {X -0.106,Y -641.271,Z 879.505,A 0.000,B 0.000,C 90.000,E1 126.916} C_DIS
LIN {X 0.242,Y -645.014,Z 879.500,A 0.000,B 0.000,C 90.000,E1 125.884} C_DIS
LIN {X 0.073,Y -647.663,Z 879.495,A 0.000,B 0.000,C 90.000,E1 125.152} C_DIS
LIN {X -0.385,Y -650.917,Z 879.490,A 0.000,B 0.000,C 90.000,E1 124.199} C_DIS
LIN {X -0.348,Y -654.707,Z 879.483,A 0.000,B 0.000,C 90.000,E1 122.959} C_DIS
LIN {X 0.194,Y -657.341,Z 879.478,A 0.000,B 0.000,C 90.000,E1 121.926} C_DIS
LIN {X -0.148,Y -658.583,Z 879.475,A 0.000,B 0.000,C 90.000,E1 121.465} C_DIS
LIN {X 0.098,Y -660.582,Z 879.469,A 0.000,B 0.000,C 90.000,E1 120.463} C_DIS
LIN {X -0.091,Y -661.924,Z 879.465,A 0.000,B 0.000,C 90.000,E1 119.745} C_DIS
LIN {X 0.059,Y -663.174,Z 879.461,A 0.000,B 0.000,C 90.000,E1 118.999} C_DIS
LIN {X 0.029,Y -666.046,Z 879.450,A 0.000,B 0.000,C 90.000,E1 117.052} C_DIS
LIN {X -0.259,Y -667.268,Z 879.445,A 0.000,B 0.000,C 90.000,E1 116.104} C_DIS
LIN {X 0.209,Y -668.029,Z 879.441,A 0.000,B 0.000,C 90.000,E1 115.335} C_DIS
LIN {X -0.365,Y -668.418,Z 879.438,A 0.000,B 0.000,C 90.000,E1 114.899} C_DIS
LIN {X 0.108,Y -668.645,Z 879.434,A 0.000,B 0.000,C 90.000,E1 114.131} C_DIS
LIN {X 0.151,Y -668.589,Z 879.431,A 0.000,B 0.000,C 90.000,E1 113.643} C_DIS
LIN {X 0.199,Y -667.875,Z 879.429,A 0.000,B 0.000,C 90.000,E1 113.153} C_DIS
LIN {X -0.260,Y -667.241,Z 879.427,A 0.000,B 0.000,C 90.000,E1 112.950} C_DIS
LIN {X -0.219,Y -664.742,Z 879.425,A 0.000,B 0.000,C 90.000,E1 112.461} C_DIS
LIN {X -0.148,Y -663.945,Z 879.424,A 0.000,B 0.000,C 90.000,E1 112.333} C_DIS
LIN {X -0.102,Y -659.074,Z 879.421,A 0.000,B 0.000,C 90.000,E1 111.844} C_DIS
LIN {X -0.015,Y -657.488,Z 879.421,A 0.000,B 0.000,C 90.000,E1 111.716} C_DIS
LIN {X 0.239,Y -655.485,Z 879.420,A 0.000,B 0.000,C 90.000,E1 111.589} C_DIS
LIN {X 0.104,Y -648.270,Z 879.418,A 0.000,B 0.000,C 90.000,E1 111.280} C_DIS
LIN {X 0.013,Y -644.634,Z 879.418,A 0.000,B 0.000,C 90.000,E1 111.153} C_DIS
LIN {X -0.269,Y -635.542,Z 879.416,A 0.000,B 0.000,C 90.000,E1 110.918} C_DIS
LIN {X -0.022,Y -618.629,Z 879.413,A 0.000,B 0.000,C 90.000,E1 110.375} C_DIS
LIN {X 0.361,Y -609.400,Z 879.411,A 0.000,B 0.000,C 90.000,E1 109.993} C_DIS
LIN {X 0.073,Y -603.340,Z 879.410,A 0.000,B 0.000,C 90.000,E1 109.758} C_DIS
LIN {X 0.000,Y -589.380,Z 879.406,A 0.000,B 0.000,C 90.000,E1 109.087} C_DIS
LIN {X 0.247,Y -585.781,Z 879.405,A 0.000,B 0.000,C 90.000,E1 108.906} C_DIS
LIN {X -0.055,Y -578.813,Z 879.404,A 0.000,B 0.000,C 90.000,E1 108.652} C_DIS
LIN {X 0.111,Y -564.774,Z 879.401,A 0.000,B 0.000,C 90.000,E1 108.181} C_DIS
LIN {X 0.070,Y -561.986,Z 879.400,A 0.000,B 0.000,C 90.000,E1 108.055} C_DIS
LIN {X 0.021,Y -559.443,Z 879.399,A 0.000,B 0.000,C 90.000,E1 107.873} C_DIS
LIN {X -0.012,Y -559.413,Z 879.399,A 0.000,B 0.000,C 90.000,E1 107.873} C_DIS
LIN {X -0.061,Y -558.219,Z 879.398,A 0.000,B 0.000,C 90.000,E1 107.638} C_DIS
LIN {X -0.053,Y -557.537,Z 879.396,A 0.000,B 0.000,C 90.000,E1 107.221} C_DIS
LIN {X 0.261,Y -558.525,Z 879.374,A 0.000,B 0.000,C 90.000,E1 103.300} C_DIS
LIN {X 0.182,Y -559.695,Z 879.363,A 0.000,B 0.000,C 90.000,E1 101.366} C_DIS
LIN {X -0.178,Y -560.664,Z 879.356,A 0.000,B 0.000,C 90.000,E1 100.018} C_DIS
LIN {X -0.007,Y -561.858,Z 879.346,A 0.000,B 0.000,C 90.000,E1 98.341} C_DIS
LIN {X -0.035,Y -562.530,Z 879.340,A 0.000,B 0.000,C 90.000,E1 97.239} C_DIS
LIN {X 0.021,Y -563.338,Z 879.333,A 0.000,B 0.000,C 90.000,E1 95.853} C_DIS
LIN {X 0.132,Y -564.115,Z 879.323,A 0.000,B 0.000,C 90.000,E1 94.188} C_DIS
LIN {X 0.158,Y -564.637,Z 879.316,A 0.000,B 0.000,C 90.000,E1 92.808} C_DIS
LIN {X -0.189,Y -565.262,Z 879.305,A 0.000,B 0.000,C 90.000,E1 90.917} C_DIS
LIN {X -0.191,Y -565.602,Z 879.297,A 0.000,B 0.000,C 90.000,E1 89.542} C_DIS
LIN {X -0.061,Y -565.890,Z 879.288,A 0.000,B 0.000,C 90.000,E1 87.879} C_DIS
LIN {X 0.183,Y -566.259,Z 879.278,A 0.000,B 0.000,C 90.000,E1 85.931} C_DIS
LIN {X 0.240,Y -566.462,Z 879.270,A 0.000,B 0.000,C 90.000,E1 84.552} C_DIS
LIN {X 0.059,Y -566.858,Z 879.259,A 0.000,B 0.000,C 90.000,E1 82.648} C_DIS
LIN {X -0.030,Y -567.377,Z 879.249,A 0.000,B 0.000,C 90.000,E1 80.735} C_DIS
LIN {X -0.008,Y -568.112,Z 879.238,A 0.000,B 0.000,C 90.000,E1 78.814} C_DIS
LIN {X -0.219,Y -568.752,Z 879.230,A 0.000,B 0.000,C 90.000,E1 77.465} C_DIS
LIN {X -0.104,Y -569.462,Z 879.221,A 0.000,B 0.000,C 90.000,E1 75.811} C_DIS
LIN {X -0.155,Y -569.989,Z 879.214,A 0.000,B 0.000,C 90.000,E1 74.448} C_DIS
LIN {X 0.133,Y -570.438,Z 879.204,A 0.000,B 0.000,C 90.000,E1 72.779} C_DIS
LIN {X 0.053,Y -570.782,Z 879.195,A 0.000,B 0.000,C 90.000,E1 71.148} C_DIS
LIN {X -0.027,Y -570.966,Z 879.186,A 0.000,B 0.000,C 90.000,E1 69.518} C_DIS
LIN {X -0.097,Y -571.120,Z 879.176,A 0.000,B 0.000,C 90.000,E1 67.614} C_DIS
LIN {X 0.094,Y -571.134,Z 879.168,A 0.000,B 0.000,C 90.000,E1 66.230} C_DIS
LIN {X 0.127,Y -571.079,Z 879.159,A 0.000,B 0.000,C 90.000,E1 64.588} C_DIS
LIN {X -0.195,Y -570.932,Z 879.151,A 0.000,B 0.000,C 90.000,E1 63.256} C_DIS
LIN {X -0.264,Y -570.668,Z 879.144,A 0.000,B 0.000,C 90.000,E1 61.897} C_DIS
LIN {X -0.234,Y -570.183,Z 879.135,A 0.000,B 0.000,C 90.000,E1 60.255} C_DIS
LIN {X 0.021,Y -569.808,Z 879.130,A 0.000,B 0.000,C 90.000,E1 59.410} C_DIS
LIN {X 0.010,Y -569.003,Z 879.122,A 0.000,B 0.000,C 90.000,E1 58.043} C_DIS
LIN {X -0.243,Y -568.399,Z 879.118,A 0.000,B 0.000,C 90.000,E1 57.248} C_DIS
LIN {X -0.316,Y -567.970,Z 879.115,A 0.000,B 0.000,C 90.000,E1 56.707} C_DIS
LIN {X -0.160,Y -566.843,Z 879.109,A 0.000,B 0.000,C 90.000,E1 55.595} C_DIS
LIN {X -0.133,Y -565.930,Z 879.104,A 0.000,B 0.000,C 90.000,E1 54.769} C_DIS
LIN {X 0.210,Y -564.871,Z 879.100,A 0.000,B 0.000,C 90.000,E1 53.909} C_DIS
LIN {X -0.138,Y -563.296,Z 879.094,A 0.000,B 0.000,C 90.000,E1 52.844} C_DIS
LIN {X -0.163,Y -561.535,Z 879.087,A 0.000,B 0.000,C 90.000,E1 51.743} C_DIS
LIN {X -0.212,Y -559.345,Z 879.081,A 0.000,B 0.000,C 90.000,E1 50.642} C_DIS
LIN {X -0.036,Y -558.193,Z 879.078,A 0.000,B 0.000,C 90.000,E1 50.070} C_DIS
LIN {X 0.143,Y -556.081,Z 879.074,A 0.000,B 0.000,C 90.000,E1 49.218} C_DIS
LIN {X -0.063,Y -553.630,Z 879.069,A 0.000,B 0.000,C 90.000,E1 48.405} C_DIS
LIN {X 0.016,Y -551.865,Z 879.066,A 0.000,B 0.000,C 90.000,E1 47.838} C_DIS
LIN {X 0.170,Y -547.825,Z 879.060,A 0.000,B 0.000,C 90.000,E1 46.701} C_DIS
LIN {X -0.193,Y -546.791,Z 879.058,A 0.000,B 0.000,C 90.000,E1 46.458} C_DIS
LIN {X 0.240,Y -543.305,Z 879.053,A 0.000,B 0.000,C 90.000,E1 45.567} C_DIS
LIN {X 0.250,Y -540.797,Z 879.050,A 0.000,B 0.000,C 90.000,E1 45.000} C_DIS
LIN {X -0.337,Y -537.259,Z 879.046,A 0.000,B 0.000,C 90.000,E1 44.352} C_DIS
LIN {X 0.016,Y -534.174,Z 879.043,A 0.000,B 0.000,C 90.000,E1 43.743} C_DIS
LIN {X 0.130,Y -529.927,Z 879.039,A 0.000,B 0.000,C 90.000,E1 43.014} C_DIS
LIN {X 0.038,Y -526.355,Z 879.036,A 0.000,B 0.000,C 90.000,E1 42.447} C_DIS
LIN {X 0.307,Y -522.545,Z 879.033,A 0.000,B 0.000,C 90.000,E1 41.838} C_DIS
LIN {X 0.012,Y -519.589,Z 879.030,A 0.000,B 0.000,C 90.000,E1 41.434} C_DIS
LIN {X 0.017,Y -512.001,Z 879.025,A 0.000,B 0.000,C 90.000,E1 40.415} C_DIS
LIN {X -0.089,Y -507.379,Z 879.021,A 0.000,B 0.000,C 90.000,E1 39.850} C_DIS
LIN {X -0.106,Y -502.420,Z 879.018,A 0.000,B 0.000,C 90.000,E1 39.277} C_DIS
LIN {X -0.071,Y -498.478,Z 879.016,A 0.000,B 0.000,C 90.000,E1 38.830} C_DIS
LIN {X -0.045,Y -490.195,Z 879.011,A 0.000,B 0.000,C 90.000,E1 37.971} C_DIS
LIN {X -0.078,Y -482.986,Z 879.007,A 0.000,B 0.000,C 90.000,E1 37.282} C_DIS
LIN {X 0.189,Y -475.526,Z 879.003,A 0.000,B 0.000,C 90.000,E1 36.583} C_DIS
LIN {X -0.190,Y -464.969,Z 878.998,A 0.000,B 0.000,C 90.000,E1 35.724} C_DIS
LIN {X 0.023,Y -454.114,Z 878.994,A 0.000,B 0.000,C 90.000,E1 34.818} C_DIS
LIN {X -0.272,Y -443.223,Z 878.989,A 0.000,B 0.000,C 90.000,E1 33.992} C_DIS
LIN {X 0.158,Y -426.098,Z 878.981,A 0.000,B 0.000,C 90.000,E1 32.546} C_DIS
LIN {X 0.219,Y -408.042,Z 878.972,A 0.000,B 0.000,C 90.000,E1 30.924} C_DIS
LIN {X -0.119,Y -400.885,Z 878.968,A 0.000,B 0.000,C 90.000,E1 30.256} C_DIS
LIN {X -0.040,Y -397.024,Z 878.966,A 0.000,B 0.000,C 90.000,E1 29.795} C_DIS
LIN {X 0.073,Y -395.617,Z 878.965,A 0.000,B 0.000,C 90.000,E1 29.617} C_DIS
LIN {X -0.040,Y -393.998,Z 878.963,A 0.000,B 0.000,C 90.000,E1 29.411} C_DIS
LIN {X -0.043,Y -392.619,Z 878.962,A 0.000,B 0.000,C 90.000,E1 29.155} C_DIS
LIN {X -0.142,Y -390.885,Z 878.960,A 0.000,B 0.000,C 90.000,E1 28.743} C_DIS
LIN {X -0.135,Y -390.468,Z 878.959,A 0.000,B 0.000,C 90.000,E1 28.565} C_DIS
LIN {X -0.098,Y -389.522,Z 878.956,A 0.000,B 0.000,C 90.000,E1 28.025} C_DIS
LIN {X 0.096,Y -389.205,Z 878.953,A 0.000,B 0.000,C 90.000,E1 27.462} C_DIS
LIN {X -0.037,Y -389.363,Z 878.947,A 0.000,B 0.000,C 90.000,E1 26.411} C_DIS
LIN {X -0.081,Y -391.373,Z 878.931,A 0.000,B 0.000,C 90.000,E1 23.567} C_DIS
LIN {X 0.040,Y -394.454,Z 878.913,A 0.000,B 0.000,C 90.000,E1 20.355} C_DIS
LIN {X 0.170,Y -397.549,Z 878.897,A 0.000,B 0.000,C 90.000,E1 17.511} C_DIS
LIN {X 0.007,Y -400.118,Z 878.886,A 0.000,B 0.000,C 90.000,E1 15.426} C_DIS
LIN {X -0.198,Y -402.909,Z 878.874,A 0.000,B 0.000,C 90.000,E1 13.355} C_DIS
LIN {X -0.030,Y -406.405,Z 878.861,A 0.000,B 0.000,C 90.000,E1 10.894} C_DIS
LIN {X 0.116,Y -410.807,Z 878.845,A 0.000,B 0.000,C 90.000,E1 8.106} C_DIS
LIN {X -0.161,Y -415.026,Z 878.832,A 0.000,B 0.000,C 90.000,E1 5.739} C_DIS
LIN {X 0.065,Y -420.239,Z 878.817,A 0.000,B 0.000,C 90.000,E1 2.980} C_DIS
LIN {X 0.161,Y -427.345,Z 878.799,A 0.000,B 0.000,C 90.000,E1 359.771} C_DIS
LIN {X -0.117,Y -433.869,Z 878.784,A 0.000,B 0.000,C 90.000,E1 357.135} C_DIS
LIN {X -0.147,Y -437.236,Z 878.777,A 0.000,B 0.000,C 90.000,E1 355.812} C_DIS
LIN {X 0.080,Y -439.252,Z 878.773,A 0.000,B 0.000,C 90.000,E1 355.122} C_DIS
LIN {X -0.207,Y -441.319,Z 878.770,A 0.000,B 0.000,C 90.000,E1 354.666} C_DIS
LIN {X 0.107,Y -443.426,Z 878.768,A 0.000,B 0.000,C 90.000,E1 354.261} C_DIS
LIN {X 0.163,Y -444.472,Z 878.767,A 0.000,B 0.000,C 90.000,E1 354.090} C_DIS
LIN {X -0.178,Y -446.183,Z 878.766,A 0.000,B 0.000,C 90.000,E1 353.970} C_DIS
LIN {X -0.211,Y -448.975,Z 878.765,A 0.000,B 0.000,C 90.000,E1 353.742} C_DIS
LIN {X 0.062,Y -454.665,Z 878.763,A 0.000,B 0.000,C 90.000,E1 353.394} C_DIS
LIN {X -0.175,Y -469.666,Z 878.760,A 0.000,B 0.000,C 90.000,E1 352.761} C_DIS
LIN {X 0.062,Y -476.369,Z 878.758,A 0.000,B 0.000,C 90.000,E1 352.413} C_DIS
LIN {X -0.030,Y -486.209,Z 878.755,A 0.000,B 0.000,C 90.000,E1 351.894} C_DIS
LIN {X -0.036,Y -497.328,Z 878.751,A 0.000,B 0.000,C 90.000,E1 351.254} C_DIS
LIN {X -0.167,Y -506.890,Z 878.748,A 0.000,B 0.000,C 90.000,E1 350.679} C_DIS
LIN {X 0.027,Y -516.325,Z 878.745,A 0.000,B 0.000,C 90.000,E1 350.038} C_DIS
LIN {X -0.004,Y -525.512,Z 878.741,A 0.000,B 0.000,C 90.000,E1 349.398} C_DIS
LIN {X 0.263,Y -531.565,Z 878.739,A 0.000,B 0.000,C 90.000,E1 348.926} C_DIS
LIN {X 0.306,Y -538.748,Z 878.735,A 0.000,B 0.000,C 90.000,E1 348.342} C_DIS
LIN {X 0.034,Y -545.818,Z 878.732,A 0.000,B 0.000,C 90.000,E1 347.757} C_DIS
LIN {X -0.021,Y -555.155,Z 878.727,A 0.000,B 0.000,C 90.000,E1 346.881} C_DIS
LIN {X -0.105,Y -561.514,Z 878.723,A 0.000,B 0.000,C 90.000,E1 346.228} C_DIS
LIN {X -0.275,Y -566.418,Z 878.720,A 0.000,B 0.000,C 90.000,E1 345.700} C_DIS
LIN {X -0.055,Y -572.215,Z 878.717,A 0.000,B 0.000,C 90.000,E1 344.991} C_DIS
LIN {X 0.122,Y -578.645,Z 878.712,A 0.000,B 0.000,C 90.000,E1 344.157} C_DIS
LIN {X -0.104,Y -583.664,Z 878.708,A 0.000,B 0.000,C 90.000,E1 343.504} C_DIS
LIN {X 0.193,Y -589.225,Z 878.704,A 0.000,B 0.000,C 90.000,E1 342.670} C_DIS
LIN {X 0.167,Y -594.308,Z 878.699,A 0.000,B 0.000,C 90.000,E1 341.873} C_DIS
LIN {X 0.064,Y -598.299,Z 878.696,A 0.000,B 0.000,C 90.000,E1 341.221} C_DIS
LIN {X -0.149,Y -604.274,Z 878.690,A 0.000,B 0.000,C 90.000,E1 340.188} C_DIS
LIN {X -0.315,Y -610.583,Z 878.683,A 0.000,B 0.000,C 90.000,E1 339.028} C_DIS
LIN {X -0.147,Y -615.897,Z 878.678,A 0.000,B 0.000,C 90.000,E1 337.975} C_DIS
LIN {X 0.104,Y -620.295,Z 878.673,A 0.000,B 0.000,C 90.000,E1 337.050} C_DIS
LIN {X -0.167,Y -625.043,Z 878.667,A 0.000,B 0.000,C 90.000,E1 336.049} C_DIS
LIN {X -0.138,Y -628.423,Z 878.663,A 0.000,B 0.000,C 90.000,E1 335.281} C_DIS
LIN {X -0.312,Y -632.542,Z 878.657,A 0.000,B 0.000,C 90.000,E1 334.280} C_DIS
LIN {X -0.114,Y -637.372,Z 878.650,A 0.000,B 0.000,C 90.000,E1 332.999} C_DIS
LIN {X 0.101,Y -640.945,Z 878.644,A 0.000,B 0.000,C 90.000,E1 331.975} C_DIS
LIN {X 0.106,Y -644.260,Z 878.639,A 0.000,B 0.000,C 90.000,E1 330.973} C_DIS
LIN {X -0.144,Y -649.607,Z 878.629,A 0.000,B 0.000,C 90.000,E1 329.253} C_DIS
LIN {X 0.169,Y -653.751,Z 878.621,A 0.000,B 0.000,C 90.000,E1 327.740} C_DIS
LIN {X 0.150,Y -656.273,Z 878.615,A 0.000,B 0.000,C 90.000,E1 326.755} C_DIS
LIN {X -0.191,Y -658.519,Z 878.610,A 0.000,B 0.000,C 90.000,E1 325.801} C_DIS
LIN {X -0.037,Y -660.866,Z 878.603,A 0.000,B 0.000,C 90.000,E1 324.562} C_DIS
LIN {X 0.044,Y -662.455,Z 878.598,A 0.000,B 0.000,C 90.000,E1 323.577} C_DIS
LIN {X 0.017,Y -663.891,Z 878.592,A 0.000,B 0.000,C 90.000,E1 322.603} C_DIS
LIN {X -0.360,Y -664.823,Z 878.588,A 0.000,B 0.000,C 90.000,E1 321.904} C_DIS
LIN {X -0.279,Y -666.487,Z 878.580,A 0.000,B 0.000,C 90.000,E1 320.436} C_DIS
LIN {X -0.237,Y -667.548,Z 878.575,A 0.000,B 0.000,C 90.000,E1 319.461} C_DIS
LIN {X -0.182,Y -668.906,Z 878.568,A 0.000,B 0.000,C 90.000,E1 318.243} C_DIS
LIN {X -0.081,Y -670.921,Z 878.557,A 0.000,B 0.000,C 90.000,E1 316.296} C_DIS
LIN {X -0.002,Y -672.329,Z 878.550,A 0.000,B 0.000,C 90.000,E1 315.081} C_DIS
LIN {X 0.058,Y -673.054,Z 878.546,A 0.000,B 0.000,C 90.000,E1 314.352} C_DIS
LIN {X -0.247,Y -674.730,Z 878.537,A 0.000,B 0.000,C 90.000,E1 312.690} C_DIS
LIN {X 0.350,Y -675.662,Z 878.532,A 0.000,B 0.000,C 90.000,E1 311.676} C_DIS
LIN {X 0.000,Y -676.495,Z 878.526,A 0.000,B 0.000,C 90.000,E1 310.744} C_DIS
LIN {X -0.103,Y -677.926,Z 878.517,A 0.000,B 0.000,C 90.000,E1 309.072} C_DIS
LIN {X -0.312,Y -678.877,Z 878.510,A 0.000,B 0.000,C 90.000,E1 307.890} C_DIS
LIN {X 0.027,Y -679.806,Z 878.504,A 0.000,B 0.000,C 90.000,E1 306.664} C_DIS
LIN {X -0.022,Y -680.649,Z 878.497,A 0.000,B 0.000,C 90.000,E1 305.471} C_DIS
LIN {X -0.058,Y -681.496,Z 878.489,A 0.000,B 0.000,C 90.000,E1 304.040} C_DIS
LIN {X 0.103,Y -682.299,Z 878.482,A 0.000,B 0.000,C 90.000,E1 302.832} C_DIS
LIN {X 0.289,Y -683.934,Z 878.471,A 0.000,B 0.000,C 90.000,E1 300.669} C_DIS
LIN {X -0.392,Y -685.572,Z 878.460,A 0.000,B 0.000,C 90.000,E1 298.821} C_DIS
LIN {X -0.217,Y -687.824,Z 878.448,A 0.000,B 0.000,C 90.000,E1 296.668} C_DIS
LIN {X 0.234,Y -689.478,Z 878.440,A 0.000,B 0.000,C 90.000,E1 295.207} C_DIS
LIN {X 0.248,Y -690.337,Z 878.435,A 0.000,B 0.000,C 90.000,E1 294.259} C_DIS
LIN {X 0.035,Y -690.743,Z 878.431,A 0.000,B 0.000,C 90.000,E1 293.567} C_DIS
LIN {X -0.006,Y -690.794,Z 878.430,A 0.000,B 0.000,C 90.000,E1 293.334} C_DIS
LIN {X 0.191,Y -690.356,Z 878.427,A 0.000,B 0.000,C 90.000,E1 292.845} C_DIS
LIN {X -0.214,Y -689.878,Z 878.426,A 0.000,B 0.000,C 90.000,E1 292.642} C_DIS
LIN {X -0.020,Y -688.150,Z 878.423,A 0.000,B 0.000,C 90.000,E1 292.153} C_DIS
LIN {X 0.091,Y -687.567,Z 878.422,A 0.000,B 0.000,C 90.000,E1 292.025} C_DIS
LIN {X 0.202,Y -686.726,Z 878.422,A 0.000,B 0.000,C 90.000,E1 291.897} C_DIS
LIN {X 0.310,Y -685.478,Z 878.421,A 0.000,B 0.000,C 90.000,E1 291.770} C_DIS
LIN {X 0.235,Y -679.553,Z 878.419,A 0.000,B 0.000,C 90.000,E1 291.354} C_DIS
LIN {X -0.079,Y -677.568,Z 878.418,A 0.000,B 0.000,C 90.000,E1 291.280} C_DIS
LIN {X -0.181,Y -668.701,Z 878.417,A 0.000,B 0.000,C 90.000,E1 291.025} C_DIS
LIN {X 0.362,Y -661.513,Z 878.416,A 0.000,B 0.000,C 90.000,E1 290.791} C_DIS
LIN {X 0.214,Y -659.599,Z 878.415,A 0.000,B 0.000,C 90.000,E1 290.737} C_DIS
LIN {X -0.254,Y -654.699,Z 878.414,A 0.000,B 0.000,C 90.000,E1 290.556} C_DIS
LIN {X -0.354,Y -653.299,Z 878.413,A 0.000,B 0.000,C 90.000,E1 290.429} C_DIS
LIN {X 0.215,Y -653.278,Z 878.413,A 0.000,B 0.000,C 90.000,E1 290.375} C_DIS
LIN {X -0.352,Y -652.979,Z 878.412,A 0.000,B 0.000,C 90.000,E1 290.248} C_DIS
LIN {X -0.174,Y -653.309,Z 878.411,A 0.000,B 0.000,C 90.000,E1 290.047} C_DIS
LIN {X 0.305,Y -654.017,Z 878.410,A 0.000,B 0.000,C 90.000,E1 289.758} C_DIS
LIN {X -0.095,Y -659.156,Z 878.404,A 0.000,B 0.000,C 90.000,E1 288.779} C_DIS
LIN {X -0.164,Y -663.650,Z 878.400,A 0.000,B 0.000,C 90.000,E1 287.928} C_DIS
LIN {X 0.191,Y -667.141,Z 878.396,A 0.000,B 0.000,C 90.000,E1 287.166} C_DIS
LIN {X 0.223,Y -669.204,Z 878.393,A 0.000,B 0.000,C 90.000,E1 286.677} C_DIS
LIN {X 0.005,Y -671.826,Z 878.389,A 0.000,B 0.000,C 90.000,E1 285.969} C_DIS
LIN {X -0.004,Y -673.912,Z 878.385,A 0.000,B 0.000,C 90.000,E1 285.245} C_DIS
LIN {X -0.119,Y -675.054,Z 878.382,A 0.000,B 0.000,C 90.000,E1 284.773} C_DIS
LIN {X -0.277,Y -676.413,Z 878.378,A 0.000,B 0.000,C 90.000,E1 284.064} C_DIS
LIN {X 0.283,Y -677.163,Z 878.375,A 0.000,B 0.000,C 90.000,E1 283.536} C_DIS
LIN {X 0.147,Y -678.014,Z 878.371,A 0.000,B 0.000,C 90.000,E1 282.827} C_DIS
LIN {X 0.014,Y -678.630,Z 878.367,A 0.000,B 0.000,C 90.000,E1 282.119} C_DIS
LIN {X -0.030,Y -678.801,Z 878.366,A 0.000,B 0.000,C 90.000,E1 281.883} C_DIS
LIN {X -0.254,Y -678.907,Z 878.363,A 0.000,B 0.000,C 90.000,E1 281.422} C_DIS
LIN {X 0.279,Y -678.578,Z 878.359,A 0.000,B 0.000,C 90.000,E1 280.658} C_DIS
LIN {X 0.063,Y -678.133,Z 878.357,A 0.000,B 0.000,C 90.000,E1 280.197} C_DIS
LIN {X -0.036,Y -677.396,Z 878.354,A 0.000,B 0.000,C 90.000,E1 279.726} C_DIS
LIN {X -0.254,Y -676.329,Z 878.351,A 0.000,B 0.000,C 90.000,E1 279.265} C_DIS
LIN {X 0.192,Y -674.970,Z 878.349,A 0.000,B 0.000,C 90.000,E1 278.746} C_DIS
LIN {X 0.063,Y -673.314,Z 878.346,A 0.000,B 0.000,C 90.000,E1 278.276} C_DIS
LIN {X -0.102,Y -672.430,Z 878.345,A 0.000,B 0.000,C 90.000,E1 278.049} C_DIS
LIN {X -0.343,Y -670.330,Z 878.342,A 0.000,B 0.000,C 90.000,E1 277.587} C_DIS
LIN {X 0.065,Y -667.326,Z 878.339,A 0.000,B 0.000,C 90.000,E1 276.947} C_DIS
LIN {X -0.301,Y -663.820,Z 878.335,A 0.000,B 0.000,C 90.000,E1 276.372} C_DIS
LIN {X 0.060,Y -660.648,Z 878.333,A 0.000,B 0.000,C 90.000,E1 275.853} C_DIS
LIN {X -0.259,Y -657.054,Z 878.330,A 0.000,B 0.000,C 90.000,E1 275.391} C_DIS
LIN {X -0.005,Y -652.821,Z 878.327,A 0.000,B 0.000,C 90.000,E1 274.878} C_DIS
LIN {X 0.198,Y -646.940,Z 878.324,A 0.000,B 0.000,C 90.000,E1 274.245} C_DIS
LIN {X -0.040,Y -640.498,Z 878.320,A 0.000,B 0.000,C 90.000,E1 273.669} C_DIS
LIN {X -0.128,Y -635.049,Z 878.318,A 0.000,B 0.000,C 90.000,E1 273.212} C_DIS
LIN {X 0.039,Y -630.904,Z 878.316,A 0.000,B 0.000,C 90.000,E1 272.865} C_DIS
LIN {X 0.034,Y -623.502,Z 878.313,A 0.000,B 0.000,C 90.000,E1 272.350} C_DIS
LIN {X 0.158,Y -617.192,Z 878.311,A 0.000,B 0.000,C 90.000,E1 271.949} C_DIS
LIN {X -0.035,Y -610.545,Z 878.309,A 0.000,B 0.000,C 90.000,E1 271.604} C_DIS
LIN {X 0.118,Y -603.562,Z 878.307,A 0.000,B 0.000,C 90.000,E1 271.260} C_DIS
LIN {X 0.011,Y -596.441,Z 878.305,A 0.000,B 0.000,C 90.000,E1 270.974} C_DIS
LIN {X -0.238,Y -590.995,Z 878.304,A 0.000,B 0.000,C 90.000,E1 270.802} C_DIS
LIN {X -0.177,Y -583.455,Z 878.303,A 0.000,B 0.000,C 90.000,E1 270.573} C_DIS
LIN {X 0.188,Y -577.943,Z 878.302,A 0.000,B 0.000,C 90.000,E1 270.401} C_DIS
LIN {X 0.123,Y -571.716,Z 878.302,A 0.000,B 0.000,C 90.000,E1 270.286} C_DIS
LIN {X -0.186,Y -564.235,Z 878.301,A 0.000,B 0.000,C 90.000,E1 270.229} C_DIS
LIN {X 0.197,Y -552.854,Z 878.301,A 0.000,B 0.000,C 90.000,E1 270.115} C_DIS
LIN {X 0.231,Y -549.189,Z 878.300,A 0.000,B 0.000,C 90.000,E1 270.000} C_DIS
LIN {X 0.195,Y -549.141,Z 878.300,A 0.000,B 0.000,C 90.000,E1 270.000} C_DIS
LIN {X 0.230,Y -547.404,Z 878.299,A 0.000,B 0.000,C 90.000,E1 269.828} C_DIS
LIN {X -0.161,Y -546.723,Z 878.298,A 0.000,B 0.000,C 90.000,E1 269.714} C_DIS
LIN {X 0.134,Y -546.269,Z 878.298,A 0.000,B 0.000,C 90.000,E1 269.542} C_DIS
LIN {X -0.074,Y -545.379,Z 878.295,A 0.000,B 0.000,C 90.000,E1 269.141} C_DIS
LIN {X -0.074,Y -541.868,Z 878.273,A 0.000,B 0.000,C 90.000,E1 265.179} C_DIS
LIN {X 0.099,Y -540.938,Z 878.265,A 0.000,B 0.000,C 90.000,E1 263.742} C_DIS
LIN {X 0.240,Y -540.119,Z 878.259,A 0.000,B 0.000,C 90.000,E1 262.591} C_DIS
LIN {X -0.099,Y -539.056,Z 878.253,A 0.000,B 0.000,C 90.000,E1 261.489} C_DIS
LIN {X 0.147,Y -537.627,Z 878.245,A 0.000,B 0.000,C 90.000,E1 260.038} C_DIS
LIN {X -0.004,Y -535.849,Z 878.235,A 0.000,B 0.000,C 90.000,E1 258.342} C_DIS
LIN {X 0.225,Y -534.607,Z 878.229,A 0.000,B 0.000,C 90.000,E1 257.173} C_DIS
LIN {X 0.080,Y -532.821,Z 878.221,A 0.000,B 0.000,C 90.000,E1 255.755} C_DIS
LIN {X 0.109,Y -530.355,Z 878.210,A 0.000,B 0.000,C 90.000,E1 253.740} C_DIS
LIN {X -0.293,Y -527.957,Z 878.199,A 0.000,B 0.000,C 90.000,E1 251.764} C_DIS
LIN {X -0.096,Y -525.708,Z 878.189,A 0.000,B 0.000,C 90.000,E1 250.007} C_DIS
LIN {X 0.063,Y -523.802,Z 878.181,A 0.000,B 0.000,C 90.000,E1 248.539} C_DIS
LIN {X 0.223,Y -522.060,Z 878.174,A 0.000,B 0.000,C 90.000,E1 247.358} C_DIS
LIN {X 0.030,Y -519.886,Z 878.166,A 0.000,B 0.000,C 90.000,E1 245.921} C_DIS
LIN {X 0.148,Y -517.177,Z 878.157,A 0.000,B 0.000,C 90.000,E1 244.152} C_DIS
LIN {X -0.041,Y -515.283,Z 878.150,A 0.000,B 0.000,C 90.000,E1 242.999} C_DIS
LIN {X -0.261,Y -512.200,Z 878.140,A 0.000,B 0.000,C 90.000,E1 241.257} C_DIS
LIN {X -0.053,Y -509.142,Z 878.130,A 0.000,B 0.000,C 90.000,E1 239.459} C_DIS
LIN {X 0.139,Y -507.001,Z 878.124,A 0.000,B 0.000,C 90.000,E1 238.250} C_DIS
LIN {X 0.296,Y -504.741,Z 878.117,A 0.000,B 0.000,C 90.000,E1 237.041} C_DIS
LIN {X -0.125,Y -501.722,Z 878.109,A 0.000,B 0.000,C 90.000,E1 235.595} C_DIS
LIN {X -0.190,Y -498.951,Z 878.102,A 0.000,B 0.000,C 90.000,E1 234.402} C_DIS
LIN {X 0.123,Y -494.648,Z 878.092,A 0.000,B 0.000,C 90.000,E1 232.557} C_DIS
LIN {X 0.003,Y -492.595,Z 878.087,A 0.000,B 0.000,C 90.000,E1 231.662} C_DIS
LIN {X -0.069,Y -489.018,Z 878.079,A 0.000,B 0.000,C 90.000,E1 230.150} C_DIS
LIN {X -0.105,Y -486.273,Z 878.072,A 0.000,B 0.000,C 90.000,E1 228.933} C_DIS
LIN {X -0.180,Y -483.510,Z 878.065,A 0.000,B 0.000,C 90.000,E1 227.715} C_DIS
LIN {X 0.155,Y -480.192,Z 878.056,A 0.000,B 0.000,C 90.000,E1 226.134} C_DIS
LIN {X 0.196,Y -476.081,Z 878.046,A 0.000,B 0.000,C 90.000,E1 224.271} C_DIS
LIN {X -0.189,Y -471.894,Z 878.036,A 0.000,B 0.000,C 90.000,E1 222.447} C_DIS
LIN {X -0.206,Y -467.066,Z 878.024,A 0.000,B 0.000,C 90.000,E1 220.253} C_DIS
LIN {X -0.247,Y -461.677,Z 878.009,A 0.000,B 0.000,C 90.000,E1 217.729} C_DIS
LIN {X 0.134,Y -458.331,Z 878.001,A 0.000,B 0.000,C 90.000,E1 216.091} C_DIS
LIN {X 0.009,Y -453.627,Z 877.988,A 0.000,B 0.000,C 90.000,E1 213.865} C_DIS
LIN {X 0.125,Y -448.807,Z 877.976,A 0.000,B 0.000,C 90.000,E1 211.592} C_DIS
LIN {X 0.069,Y -443.249,Z 877.961,A 0.000,B 0.000,C 90.000,E1 208.999} C_DIS
LIN {X -0.106,Y -439.621,Z 877.952,A 0.000,B 0.000,C 90.000,E1 207.385} C_DIS
LIN {X -0.113,Y -434.642,Z 877.939,A 0.000,B 0.000,C 90.000,E1 205.079} C_DIS
LIN {X -0.042,Y -430.487,Z 877.928,A 0.000,B 0.000,C 90.000,E1 203.078} C_DIS
LIN {X -0.237,Y -425.013,Z 877.913,A 0.000,B 0.000,C 90.000,E1 200.429} C_DIS
LIN {X 0.126,Y -422.257,Z 877.906,A 0.000,B 0.000,C 90.000,E1 199.033} C_DIS
LIN {X 0.083,Y -418.930,Z 877.896,A 0.000,B 0.000,C 90.000,E1 197.347} C_DIS
LIN {X -0.184,Y -416.156,Z 877.889,A 0.000,B 0.000,C 90.000,E1 196.024} C_DIS
LIN {X -0.070,Y -412.682,Z 877.879,A 0.000,B 0.000,C 90.000,E1 194.300} C_DIS
LIN {X -0.156,Y -410.027,Z 877.872,A 0.000,B 0.000,C 90.000,E1 192.939} C_DIS
LIN {X 0.020,Y -407.363,Z 877.864,A 0.000,B 0.000,C 90.000,E1 191.535} C_DIS
LIN {X 0.088,Y -404.026,Z 877.854,A 0.000,B 0.000,C 90.000,E1 189.792} C_DIS
LIN {X 0.090,Y -400.446,Z 877.845,A 0.000,B 0.000,C 90.000,E1 188.049} C_DIS
LIN {X -0.170,Y -395.048,Z 877.829,A 0.000,B 0.000,C 90.000,E1 185.277} C_DIS
LIN {X 0.080,Y -390.443,Z 877.813,A 0.000,B 0.000,C 90.000,E1 182.407} C_DIS
LIN {X -0.045,Y -387.298,Z 877.802,A 0.000,B 0.000,C 90.000,E1 180.286} C_DIS
LIN {X -0.046,Y -385.257,Z 877.794,A 0.000,B 0.000,C 90.000,E1 178.854} C_DIS
LIN {X 0.102,Y -382.041,Z 877.782,A 0.000,B 0.000,C 90.000,E1 176.674} C_DIS
LIN {X 0.199,Y -378.804,Z 877.770,A 0.000,B 0.000,C 90.000,E1 174.489} C_DIS
LIN {X 0.142,Y -375.627,Z 877.755,A 0.000,B 0.000,C 90.000,E1 171.951} C_DIS
LIN {X 0.075,Y -374.443,Z 877.747,A 0.000,B 0.000,C 90.000,E1 170.500} C_DIS
LIN {X 0.103,Y -373.881,Z 877.741,A 0.000,B 0.000,C 90.000,E1 169.398} C_DIS
LIN {X -0.131,Y -373.857,Z 877.737,A 0.000,B 0.000,C 90.000,E1 168.701} C_DIS
LIN {X 0.074,Y -374.133,Z 877.733,A 0.000,B 0.000,C 90.000,E1 167.937} C_DIS
LIN {X -0.126,Y -375.098,Z 877.727,A 0.000,B 0.000,C 90.000,E1 166.881} C_DIS
LIN {X 0.209,Y -375.550,Z 877.725,A 0.000,B 0.000,C 90.000,E1 166.464} C_DIS
LIN {X 0.068,Y -377.326,Z 877.721,A 0.000,B 0.000,C 90.000,E1 165.755} C_DIS
LIN {X -0.047,Y -378.306,Z 877.719,A 0.000,B 0.000,C 90.000,E1 165.408} C_DIS
LIN {X -0.065,Y -379.711,Z 877.717,A 0.000,B 0.000,C 90.000,E1 165.046} C_DIS
LIN {X -0.101,Y -381.037,Z 877.715,A 0.000,B 0.000,C 90.000,E1 164.755} C_DIS
LIN {X -0.106,Y -383.319,Z 877.713,A 0.000,B 0.000,C 90.000,E1 164.393} C_DIS
LIN {X -0.103,Y -384.639,Z 877.712,A 0.000,B 0.000,C 90.000,E1 164.212} C_DIS
LIN {X 0.026,Y -390.689,Z 877.709,A 0.000,B 0.000,C 90.000,E1 163.614} C_DIS
LIN {X -0.067,Y -396.078,Z 877.707,A 0.000,B 0.000,C 90.000,E1 163.268} C_DIS
LIN {X -0.197,Y -417.159,Z 877.701,A 0.000,B 0.000,C 90.000,E1 162.181} C_DIS
LIN {X -0.147,Y -420.345,Z 877.700,A 0.000,B 0.000,C 90.000,E1 162.000} C_DIS
LIN {X 0.038,Y -426.822,Z 877.698,A 0.000,B 0.000,C 90.000,E1 161.583} C_DIS
LIN {X 0.129,Y -436.094,Z 877.694,A 0.000,B 0.000,C 90.000,E1 160.913} C_DIS
LIN {X 0.160,Y -443.825,Z 877.691,A 0.000,B 0.000,C 90.000,E1 160.315} C_DIS
LIN {X 0.069,Y -449.933,Z 877.688,A 0.000,B 0.000,C 90.000,E1 159.826} C_DIS
LIN {X 0.113,Y -458.786,Z 877.684,A 0.000,B 0.000,C 90.000,E1 159.028} C_DIS
LIN {X 0.066,Y -461.652,Z 877.682,A 0.000,B 0.000,C 90.000,E1 158.773} C_DIS
LIN {X -0.198,Y -472.803,Z 877.676,A 0.000,B 0.000,C 90.000,E1 157.667} C_DIS
LIN {X -0.105,Y -482.116,Z 877.670,A 0.000,B 0.000,C 90.000,E1 156.613} C_DIS
LIN {X -0.010,Y -490.931,Z 877.664,A 0.000,B 0.000,C 90.000,E1 155.537} C_DIS
LIN {X 0.095,Y -498.043,Z 877.659,A 0.000,B 0.000,C 90.000,E1 154.613} C_DIS
LIN {X 0.165,Y -501.367,Z 877.657,A 0.000,B 0.000,C 90.000,E1 154.152} C_DIS
LIN {X -0.033,Y -508.916,Z 877.651,A 0.000,B 0.000,C 90.000,E1 153.127} C_DIS
LIN {X -0.071,Y -517.057,Z 877.644,A 0.000,B 0.000,C 90.000,E1 151.948} C_DIS
LIN {X 0.087,Y -523.143,Z 877.639,A 0.000,B 0.000,C 90.000,E1 151.051} C_DIS
LIN {X 0.261,Y -530.580,Z 877.633,A 0.000,B 0.000,C 90.000,E1 149.871} C_DIS
LIN {X -0.064,Y -538.275,Z 877.626,A 0.000,B 0.000,C 90.000,E1 148.614} C_DIS
LIN {X 0.170,Y -546.215,Z 877.618,A 0.000,B 0.000,C 90.000,E1 147.168} C_DIS
LIN {X -0.008,Y -550.932,Z 877.613,A 0.000,B 0.000,C 90.000,E1 146.342} C_DIS
LIN {X -0.138,Y -555.357,Z 877.608,A 0.000,B 0.000,C 90.000,E1 145.515} C_DIS
LIN {X -0.020,Y -560.143,Z 877.603,A 0.000,B 0.000,C 90.000,E1 144.529} C_DIS
LIN {X 0.166,Y -569.279,Z 877.593,A 0.000,B 0.000,C 90.000,E1 142.718} C_DIS
LIN {X -0.018,Y -577.823,Z 877.583,A 0.000,B 0.000,C 90.000,E1 140.964} C_DIS
LIN {X 0.280,Y -582.344,Z 877.578,A 0.000,B 0.000,C 90.000,E1 139.989} C_DIS
LIN {X -0.007,Y -587.815,Z 877.571,A 0.000,B 0.000,C 90.000,E1 138.809} C_DIS
LIN {X 0.005,Y -596.546,Z 877.561,A 0.000,B 0.000,C 90.000,E1 136.944} C_DIS
LIN {X -0.110,Y -604.694,Z 877.551,A 0.000,B 0.000,C 90.000,E1 135.243} C_DIS
LIN {X -0.211,Y -610.596,Z 877.544,A 0.000,B 0.000,C 90.000,E1 133.947} C_DIS
LIN {X 0.225,Y -616.359,Z 877.537,A 0.000,B 0.000,C 90.000,E1 132.609} C_DIS
LIN {X -0.117,Y -621.969,Z 877.530,A 0.000,B 0.000,C 90.000,E1 131.353} C_DIS
LIN {X -0.314,Y -627.274,Z 877.523,A 0.000,B 0.000,C 90.000,E1 130.092} C_DIS
LIN {X 0.110,Y -631.261,Z 877.517,A 0.000,B 0.000,C 90.000,E1 129.036} C_DIS
LIN {X 0.191,Y -635.189,Z 877.511,A 0.000,B 0.000,C 90.000,E1 128.016} C_DIS
LIN {X -0.060,Y -639.135,Z 877.506,A 0.000,B 0.000,C 90.000,E1 127.030} C_DIS
LIN {X -0.277,Y -642.038,Z 877.502,A 0.000,B 0.000,C 90.000,E1 126.297} C_DIS
LIN {X 0.048,Y -644.800,Z 877.497,A 0.000,B 0.000,C 90.000,E1 125.518} C_DIS
LIN {X -0.016,Y -648.916,Z 877.490,A 0.000,B 0.000,C 90.000,E1 124.278} C_DIS
LIN {X -0.008,Y -652.711,Z 877.484,A 0.000,B 0.000,C 90.000,E1 123.038} C_DIS
LIN {X -0.043,Y -655.393,Z 877.478,A 0.000,B 0.000,C 90.000,E1 122.054} C_DIS
LIN {X -0.294,Y -657.164,Z 877.474,A 0.000,B 0.000,C 90.000,E1 121.337} C_DIS
LIN {X -0.064,Y -659.141,Z 877.469,A 0.000,B 0.000,C 90.000,E1 120.335} C_DIS
LIN {X 0.187,Y -660.860,Z 877.463,A 0.000,B 0.000,C 90.000,E1 119.333} C_DIS
LIN {X 0.000,Y -662.057,Z 877.459,A 0.000,B 0.000,C 90.000,E1 118.615} C_DIS
LIN {X -0.199,Y -664.589,Z 877.450,A 0.000,B 0.000,C 90.000,E1 116.924} C_DIS
LIN {X 0.244,Y -666.088,Z 877.443,A 0.000,B 0.000,C 90.000,E1 115.668} C_DIS
LIN {X 0.096,Y -666.728,Z 877.439,A 0.000,B 0.000,C 90.000,E1 114.951} C_DIS
LIN {X 0.275,Y -666.993,Z 877.435,A 0.000,B 0.000,C 90.000,E1 114.207} C_DIS
LIN {X -0.300,Y -666.979,Z 877.432,A 0.000,B 0.000,C 90.000,E1 113.770} C_DIS
LIN {X 0.001,Y -666.336,Z 877.429,A 0.000,B 0.000,C 90.000,E1 113.259} C_DIS
LIN {X -0.112,Y -665.813,Z 877.428,A 0.000,B 0.000,C 90.000,E1 113.025} C_DIS
LIN {X 0.178,Y -663.489,Z 877.425,A 0.000,B 0.000,C 90.000,E1 112.514} C_DIS
LIN {X -0.005,Y -662.785,Z 877.425,A 0.000,B 0.000,C 90.000,E1 112.408} C_DIS
LIN {X 0.130,Y -660.456,Z 877.423,A 0.000,B 0.000,C 90.000,E1 112.153} C_DIS
LIN {X 0.196,Y -659.221,Z 877.422,A 0.000,B 0.000,C 90.000,E1 112.025} C_DIS
LIN {X 0.281,Y -658.205,Z 877.422,A 0.000,B 0.000,C 90.000,E1 111.897} C_DIS
LIN {X 0.121,Y -656.864,Z 877.421,A 0.000,B 0.000,C 90.000,E1 111.791} C_DIS
LIN {X -0.346,Y -654.976,Z 877.421,A 0.000,B 0.000,C 90.000,E1 111.716} C_DIS
LIN {X -0.204,Y -652.776,Z 877.420,A 0.000,B 0.000,C 90.000,E1 111.589} C_DIS
LIN {X 0.067,Y -650.862,Z 877.419,A 0.000,B 0.000,C 90.000,E1 111.482} C_DIS
LIN {X 0.312,Y -647.348,Z 877.418,A 0.000,B 0.000,C 90.000,E1 111.280} C_DIS
LIN {X -0.155,Y -641.236,Z 877.417,A 0.000,B 0.000,C 90.000,E1 111.099} C_DIS
LIN {X 0.006,Y -625.816,Z 877.415,A 0.000,B 0.000,C 90.000,E1 110.610} C_DIS
LIN {X 0.195,Y -618.891,Z 877.413,A 0.000,B 0.000,C 90.000,E1 110.375} C_DIS
LIN {X -0.221,Y -609.629,Z 877.411,A 0.000,B 0.000,C 90.000,E1 110.066} C_DIS
LIN {X 0.283,Y -603.626,Z 877.410,A 0.000,B 0.000,C 90.000,E1 109.758} C_DIS
LIN {X -0.337,Y -591.115,Z 877.407,A 0.000,B 0.000,C 90.000,E1 109.214} C_DIS
LIN {X -0.098,Y -587.797,Z 877.406,A 0.000,B 0.000,C 90.000,E1 109.033} C_DIS
LIN {X -0.108,Y -578.679,Z 877.404,A 0.000,B 0.000,C 90.000,E1 108.671} C_DIS
LIN {X 0.307,Y -566.284,Z 877.402,A 0.000,B 0.000,C 90.000,E1 108.236} C_DIS
LIN {X 0.221,Y -563.327,Z 877.401,A 0.000,B 0.000,C 90.000,E1 108.127} C_DIS
LIN {X 0.205,Y -561.942,Z 877.400,A 0.000,B 0.000,C 90.000,E1 108.055} C_DIS
LIN {X -0.251,Y -559.887,Z 877.400,A 0.000,B 0.000,C 90.000,E1 107.946} C_DIS
LIN {X 0.074,Y -558.464,Z 877.398,A 0.000,B 0.000,C 90.000,E1 107.638} C_DIS
LIN {X 0.084,Y -557.782,Z 877.396,A 0.000,B 0.000,C 90.000,E1 107.221} C_DIS
LIN {X -0.016,Y -557.984,Z 877.383,A 0.000,B 0.000,C 90.000,E1 105.009} C_DIS
LIN {X 0.006,Y -558.846,Z 877.373,A 0.000,B 0.000,C 90.000,E1 103.063} C_DIS
LIN {X -0.215,Y -559.873,Z 877.363,A 0.000,B 0.000,C 90.000,E1 101.422} C_DIS
LIN {X 0.183,Y -561.215,Z 877.353,A 0.000,B 0.000,C 90.000,E1 99.443} C_DIS
LIN {X -0.253,Y -562.190,Z 877.345,A 0.000,B 0.000,C 90.000,E1 98.106} C_DIS
LIN {X -0.051,Y -563.212,Z 877.336,A 0.000,B 0.000,C 90.000,E1 96.429} C_DIS
LIN {X -0.042,Y -563.886,Z 877.328,A 0.000,B 0.000,C 90.000,E1 95.049} C_DIS
LIN {X -0.019,Y -564.504,Z 877.320,A 0.000,B 0.000,C 90.000,E1 93.669} C_DIS
LIN {X -0.020,Y -564.964,Z 877.313,A 0.000,B 0.000,C 90.000,E1 92.293} C_DIS
LIN {X 0.098,Y -565.505,Z 877.304,A 0.000,B 0.000,C 90.000,E1 90.630} C_DIS
LIN {X 0.101,Y -565.803,Z 877.296,A 0.000,B 0.000,C 90.000,E1 89.255} C_DIS
LIN {X 0.235,Y -566.101,Z 877.287,A 0.000,B 0.000,C 90.000,E1 87.593} C_DIS
LIN {X -0.047,Y -566.472,Z 877.276,A 0.000,B 0.000,C 90.000,E1 85.698} C_DIS
LIN {X 0.125,Y -566.724,Z 877.267,A 0.000,B 0.000,C 90.000,E1 84.033} C_DIS
LIN {X -0.049,Y -567.128,Z 877.256,A 0.000,B 0.000,C 90.000,E1 82.129} C_DIS
LIN {X -0.041,Y -567.740,Z 877.246,A 0.000,B 0.000,C 90.000,E1 80.208} C_DIS
LIN {X -0.198,Y -568.789,Z 877.232,A 0.000,B 0.000,C 90.000,E1 77.757} C_DIS
LIN {X -0.217,Y -569.456,Z 877.223,A 0.000,B 0.000,C 90.000,E1 76.117} C_DIS
LIN {X 0.053,Y -570.092,Z 877.214,A 0.000,B 0.000,C 90.000,E1 74.448} C_DIS
LIN {X 0.003,Y -570.473,Z 877.206,A 0.000,B 0.000,C 90.000,E1 73.087} C_DIS
LIN {X -0.082,Y -570.832,Z 877.197,A 0.000,B 0.000,C 90.000,E1 71.456} C_DIS
LIN {X 0.188,Y -571.055,Z 877.186,A 0.000,B 0.000,C 90.000,E1 69.518} C_DIS
LIN {X 0.120,Y -571.182,Z 877.176,A 0.000,B 0.000,C 90.000,E1 67.614} C_DIS
LIN {X 0.312,Y -571.192,Z 877.168,A 0.000,B 0.000,C 90.000,E1 66.230} C_DIS
LIN {X 0.100,Y -571.115,Z 877.159,A 0.000,B 0.000,C 90.000,E1 64.613} C_DIS
LIN {X 0.025,Y -570.967,Z 877.151,A 0.000,B 0.000,C 90.000,E1 63.256} C_DIS
LIN {X -0.044,Y -570.677,Z 877.144,A 0.000,B 0.000,C 90.000,E1 61.897} C_DIS
LIN {X -0.123,Y -570.267,Z 877.136,A 0.000,B 0.000,C 90.000,E1 60.539} C_DIS
LIN {X 0.240,Y -569.780,Z 877.130,A 0.000,B 0.000,C 90.000,E1 59.410} C_DIS
LIN {X -0.073,Y -568.938,Z 877.123,A 0.000,B 0.000,C 90.000,E1 58.074} C_DIS
LIN {X -0.026,Y -568.332,Z 877.118,A 0.000,B 0.000,C 90.000,E1 57.248} C_DIS
LIN {X -0.100,Y -567.896,Z 877.115,A 0.000,B 0.000,C 90.000,E1 56.707} C_DIS
LIN {X 0.055,Y -566.732,Z 877.109,A 0.000,B 0.000,C 90.000,E1 55.595} C_DIS
LIN {X 0.195,Y -565.465,Z 877.103,A 0.000,B 0.000,C 90.000,E1 54.482} C_DIS
LIN {X -0.145,Y -563.961,Z 877.097,A 0.000,B 0.000,C 90.000,E1 53.417} C_DIS
LIN {X 0.282,Y -562.250,Z 877.091,A 0.000,B 0.000,C 90.000,E1 52.271} C_DIS
LIN {X 0.043,Y -561.335,Z 877.088,A 0.000,B 0.000,C 90.000,E1 51.743} C_DIS
LIN {X -0.010,Y -559.112,Z 877.081,A 0.000,B 0.000,C 90.000,E1 50.642} C_DIS
LIN {X 0.165,Y -557.951,Z 877.078,A 0.000,B 0.000,C 90.000,E1 50.070} C_DIS
LIN {X -0.023,Y -555.784,Z 877.074,A 0.000,B 0.000,C 90.000,E1 49.256} C_DIS
LIN {X 0.130,Y -553.323,Z 877.069,A 0.000,B 0.000,C 90.000,E1 48.405} C_DIS
LIN {X -0.164,Y -551.531,Z 877.066,A 0.000,B 0.000,C 90.000,E1 47.877} C_DIS
LIN {X -0.044,Y -547.446,Z 877.060,A 0.000,B 0.000,C 90.000,E1 46.743} C_DIS
LIN {X -0.011,Y -546.408,Z 877.058,A 0.000,B 0.000,C 90.000,E1 46.458} C_DIS
LIN {X 0.037,Y -542.840,Z 877.053,A 0.000,B 0.000,C 90.000,E1 45.607} C_DIS
LIN {X 0.041,Y -540.282,Z 877.050,A 0.000,B 0.000,C 90.000,E1 45.040} C_DIS
LIN {X -0.169,Y -536.696,Z 877.046,A 0.000,B 0.000,C 90.000,E1 44.352} C_DIS
LIN {X -0.208,Y -533.590,Z 877.043,A 0.000,B 0.000,C 90.000,E1 43.785} C_DIS
LIN {X 0.062,Y -528.407,Z 877.038,A 0.000,B 0.000,C 90.000,E1 42.894} C_DIS
LIN {X 0.188,Y -525.665,Z 877.036,A 0.000,B 0.000,C 90.000,E1 42.447} C_DIS
LIN {X 0.009,Y -519.831,Z 877.031,A 0.000,B 0.000,C 90.000,E1 41.595} C_DIS
LIN {X 0.184,Y -513.261,Z 877.026,A 0.000,B 0.000,C 90.000,E1 40.701} C_DIS
LIN {X -0.159,Y -509.831,Z 877.024,A 0.000,B 0.000,C 90.000,E1 40.297} C_DIS
LIN {X -0.130,Y -506.206,Z 877.021,A 0.000,B 0.000,C 90.000,E1 39.850} C_DIS
LIN {X -0.022,Y -502.462,Z 877.019,A 0.000,B 0.000,C 90.000,E1 39.402} C_DIS
LIN {X -0.261,Y -496.157,Z 877.015,A 0.000,B 0.000,C 90.000,E1 38.749} C_DIS
LIN {X -0.193,Y -490.665,Z 877.012,A 0.000,B 0.000,C 90.000,E1 38.177} C_DIS
LIN {X 0.146,Y -483.455,Z 877.008,A 0.000,B 0.000,C 90.000,E1 37.443} C_DIS
LIN {X 0.042,Y -476.012,Z 877.004,A 0.000,B 0.000,C 90.000,E1 36.790} C_DIS
LIN {X 0.070,Y -465.480,Z 876.999,A 0.000,B 0.000,C 90.000,E1 35.884} C_DIS
LIN {X -0.102,Y -454.581,Z 876.995,A 0.000,B 0.000,C 90.000,E1 35.025} C_DIS
LIN {X -0.103,Y -446.774,Z 876.991,A 0.000,B 0.000,C 90.000,E1 34.405} C_DIS
LIN {X 0.190,Y -426.735,Z 876.982,A 0.000,B 0.000,C 90.000,E1 32.752} C_DIS
LIN {X -0.078,Y -408.599,Z 876.973,A 0.000,B 0.000,C 90.000,E1 31.180} C_DIS
LIN {X -0.193,Y -399.997,Z 876.968,A 0.000,B 0.000,C 90.000,E1 30.335} C_DIS
LIN {X -0.088,Y -394.675,Z 876.965,A 0.000,B 0.000,C 90.000,E1 29.667} C_DIS
LIN {X 0.129,Y -392.587,Z 876.963,A 0.000,B 0.000,C 90.000,E1 29.283} C_DIS
LIN {X -0.198,Y -391.024,Z 876.961,A 0.000,B 0.000,C 90.000,E1 28.949} C_DIS
LIN {X -0.005,Y -390.443,Z 876.960,A 0.000,B 0.000,C 90.000,E1 28.743} C_DIS
LIN {X -0.152,Y -389.593,Z 876.957,A 0.000,B 0.000,C 90.000,E1 28.231} C_DIS
LIN {X -0.070,Y -389.240,Z 876.952,A 0.000,B 0.000,C 90.000,E1 27.308} C_DIS
LIN {X -0.032,Y -389.607,Z 876.946,A 0.000,B 0.000,C 90.000,E1 26.232} C_DIS
LIN {X 0.105,Y -391.396,Z 876.932,A 0.000,B 0.000,C 90.000,E1 23.718} C_DIS
LIN {X -0.172,Y -394.020,Z 876.916,A 0.000,B 0.000,C 90.000,E1 20.918} C_DIS
LIN {X -0.116,Y -395.870,Z 876.906,A 0.000,B 0.000,C 90.000,E1 19.141} C_DIS
LIN {X -0.133,Y -398.739,Z 876.893,A 0.000,B 0.000,C 90.000,E1 16.677} C_DIS
LIN {X 0.101,Y -401.838,Z 876.879,A 0.000,B 0.000,C 90.000,E1 14.189} C_DIS
LIN {X -0.061,Y -405.262,Z 876.865,A 0.000,B 0.000,C 90.000,E1 11.771} C_DIS
LIN {X 0.137,Y -410.088,Z 876.848,A 0.000,B 0.000,C 90.000,E1 8.624} C_DIS
LIN {X -0.126,Y -414.854,Z 876.833,A 0.000,B 0.000,C 90.000,E1 5.910} C_DIS
LIN {X 0.068,Y -420.038,Z 876.818,A 0.000,B 0.000,C 90.000,E1 3.154} C_DIS
LIN {X 0.162,Y -427.474,Z 876.799,A 0.000,B 0.000,C 90.000,E1 359.771} C_DIS
LIN {X -0.113,Y -434.000,Z 876.784,A 0.000,B 0.000,C 90.000,E1 357.135} C_DIS
LIN {X -0.047,Y -438.263,Z 876.775,A 0.000,B 0.000,C 90.000,E1 355.469} C_DIS
LIN {X 0.137,Y -439.864,Z 876.772,A 0.000,B 0.000,C 90.000,E1 354.951} C_DIS
LIN {X -0.106,Y -441.897,Z 876.769,A 0.000,B 0.000,C 90.000,E1 354.489} C_DIS
LIN {X 0.106,Y -444.899,Z 876.767,A 0.000,B 0.000,C 90.000,E1 353.970} C_DIS
LIN {X -0.107,Y -449.857,Z 876.764,A 0.000,B 0.000,C 90.000,E1 353.571} C_DIS
LIN {X 0.159,Y -455.752,Z 876.763,A 0.000,B 0.000,C 90.000,E1 353.223} C_DIS
LIN {X -0.002,Y -468.135,Z 876.760,A 0.000,B 0.000,C 90.000,E1 352.704} C_DIS
LIN {X -0.145,Y -474.634,Z 876.758,A 0.000,B 0.000,C 90.000,E1 352.413} C_DIS
LIN {X -0.151,Y -484.466,Z 876.755,A 0.000,B 0.000,C 90.000,E1 351.894} C_DIS
LIN {X -0.151,Y -492.537,Z 876.752,A 0.000,B 0.000,C 90.000,E1 351.432} C_DIS
LIN {X -0.099,Y -502.169,Z 876.749,A 0.000,B 0.000,C 90.000,E1 350.849} C_DIS
LIN {X 0.125,Y -511.679,Z 876.746,A 0.000,B 0.000,C 90.000,E1 350.218} C_DIS
LIN {X -0.289,Y -520.967,Z 876.742,A 0.000,B 0.000,C 90.000,E1 349.634} C_DIS
LIN {X 0.134,Y -530.111,Z 876.739,A 0.000,B 0.000,C 90.000,E1 348.926} C_DIS
LIN {X 0.206,Y -535.932,Z 876.736,A 0.000,B 0.000,C 90.000,E1 348.465} C_DIS
LIN {X 0.016,Y -544.416,Z 876.732,A 0.000,B 0.000,C 90.000,E1 347.757} C_DIS
LIN {X 0.286,Y -549.876,Z 876.729,A 0.000,B 0.000,C 90.000,E1 347.229} C_DIS
LIN {X -0.087,Y -555.269,Z 876.726,A 0.000,B 0.000,C 90.000,E1 346.756} C_DIS
LIN {X -0.294,Y -561.614,Z 876.723,A 0.000,B 0.000,C 90.000,E1 346.117} C_DIS
LIN {X 0.227,Y -566.515,Z 876.720,A 0.000,B 0.000,C 90.000,E1 345.519} C_DIS
LIN {X -0.096,Y -572.327,Z 876.716,A 0.000,B 0.000,C 90.000,E1 344.866} C_DIS
LIN {X 0.085,Y -578.780,Z 876.711,A 0.000,B 0.000,C 90.000,E1 344.031} C_DIS
LIN {X -0.050,Y -582.854,Z 876.708,A 0.000,B 0.000,C 90.000,E1 343.504} C_DIS
LIN {X -0.073,Y -587.636,Z 876.705,A 0.000,B 0.000,C 90.000,E1 342.834} C_DIS
LIN {X 0.269,Y -592.859,Z 876.700,A 0.000,B 0.000,C 90.000,E1 342.000} C_DIS
LIN {X 0.154,Y -596.923,Z 876.697,A 0.000,B 0.000,C 90.000,E1 341.348} C_DIS
LIN {X -0.079,Y -602.988,Z 876.691,A 0.000,B 0.000,C 90.000,E1 340.315} C_DIS
LIN {X 0.011,Y -607.979,Z 876.686,A 0.000,B 0.000,C 90.000,E1 339.390} C_DIS
LIN {X 0.193,Y -612.142,Z 876.681,A 0.000,B 0.000,C 90.000,E1 338.592} C_DIS
LIN {X -0.181,Y -617.399,Z 876.675,A 0.000,B 0.000,C 90.000,E1 337.592} C_DIS
LIN {X 0.093,Y -621.765,Z 876.670,A 0.000,B 0.000,C 90.000,E1 336.666} C_DIS
LIN {X -0.160,Y -625.872,Z 876.665,A 0.000,B 0.000,C 90.000,E1 335.793} C_DIS
LIN {X -0.121,Y -629.204,Z 876.661,A 0.000,B 0.000,C 90.000,E1 335.025} C_DIS
LIN {X -0.284,Y -633.264,Z 876.656,A 0.000,B 0.000,C 90.000,E1 334.024} C_DIS
LIN {X -0.123,Y -637.166,Z 876.650,A 0.000,B 0.000,C 90.000,E1 332.999} C_DIS
LIN {X 0.091,Y -640.765,Z 876.644,A 0.000,B 0.000,C 90.000,E1 331.975} C_DIS
LIN {X 0.093,Y -644.115,Z 876.639,A 0.000,B 0.000,C 90.000,E1 330.973} C_DIS
LIN {X -0.014,Y -648.748,Z 876.631,A 0.000,B 0.000,C 90.000,E1 329.488} C_DIS
LIN {X 0.096,Y -651.628,Z 876.625,A 0.000,B 0.000,C 90.000,E1 328.486} C_DIS
LIN {X 0.042,Y -654.377,Z 876.620,A 0.000,B 0.000,C 90.000,E1 327.502} C_DIS
LIN {X 0.228,Y -656.865,Z 876.614,A 0.000,B 0.000,C 90.000,E1 326.501} C_DIS
LIN {X 0.260,Y -659.058,Z 876.609,A 0.000,B 0.000,C 90.000,E1 325.515} C_DIS
LIN {X -0.112,Y -661.378,Z 876.602,A 0.000,B 0.000,C 90.000,E1 324.322} C_DIS
LIN {X -0.016,Y -662.969,Z 876.596,A 0.000,B 0.000,C 90.000,E1 323.336} C_DIS
LIN {X 0.093,Y -664.375,Z 876.591,A 0.000,B 0.000,C 90.000,E1 322.351} C_DIS
LIN {X 0.123,Y -665.300,Z 876.587,A 0.000,B 0.000,C 90.000,E1 321.618} C_DIS
LIN {X 0.212,Y -666.997,Z 876.579,A 0.000,B 0.000,C 90.000,E1 320.150} C_DIS
LIN {X 0.255,Y -668.360,Z 876.572,A 0.000,B 0.000,C 90.000,E1 318.933} C_DIS
LIN {X -0.174,Y -669.637,Z 876.565,A 0.000,B 0.000,C 90.000,E1 317.757} C_DIS
LIN {X -0.014,Y -672.349,Z 876.552,A 0.000,B 0.000,C 90.000,E1 315.324} C_DIS
LIN {X 0.046,Y -673.142,Z 876.548,A 0.000,B 0.000,C 90.000,E1 314.595} C_DIS
LIN {X -0.206,Y -675.232,Z 876.536,A 0.000,B 0.000,C 90.000,E1 312.447} C_DIS
LIN {X -0.002,Y -676.595,Z 876.528,A 0.000,B 0.000,C 90.000,E1 310.987} C_DIS
LIN {X -0.073,Y -678.200,Z 876.517,A 0.000,B 0.000,C 90.000,E1 309.072} C_DIS
LIN {X -0.279,Y -679.155,Z 876.510,A 0.000,B 0.000,C 90.000,E1 307.890} C_DIS
LIN {X 0.065,Y -680.090,Z 876.504,A 0.000,B 0.000,C 90.000,E1 306.664} C_DIS
LIN {X 0.021,Y -680.920,Z 876.497,A 0.000,B 0.000,C 90.000,E1 305.471} C_DIS
LIN {X -0.007,Y -681.658,Z 876.490,A 0.000,B 0.000,C 90.000,E1 304.278} C_DIS
LIN {X 0.156,Y -682.602,Z 876.483,A 0.000,B 0.000,C 90.000,E1 302.832} C_DIS
LIN {X 0.146,Y -684.027,Z 876.472,A 0.000,B 0.000,C 90.000,E1 300.924} C_DIS
LIN {X -0.372,Y -685.207,Z 876.464,A 0.000,B 0.000,C 90.000,E1 299.539} C_DIS
LIN {X -0.043,Y -686.794,Z 876.455,A 0.000,B 0.000,C 90.000,E1 297.847} C_DIS
LIN {X 0.088,Y -688.355,Z 876.447,A 0.000,B 0.000,C 90.000,E1 296.411} C_DIS
LIN {X 0.318,Y -689.713,Z 876.440,A 0.000,B 0.000,C 90.000,E1 295.207} C_DIS
LIN {X 0.051,Y -690.580,Z 876.435,A 0.000,B 0.000,C 90.000,E1 294.283} C_DIS
LIN {X -0.109,Y -690.878,Z 876.432,A 0.000,B 0.000,C 90.000,E1 293.823} C_DIS
LIN {X 0.084,Y -691.035,Z 876.430,A 0.000,B 0.000,C 90.000,E1 293.334} C_DIS
LIN {X -0.355,Y -690.545,Z 876.427,A 0.000,B 0.000,C 90.000,E1 292.898} C_DIS
LIN {X -0.122,Y -690.100,Z 876.426,A 0.000,B 0.000,C 90.000,E1 292.642} C_DIS
LIN {X 0.107,Y -689.255,Z 876.424,A 0.000,B 0.000,C 90.000,E1 292.386} C_DIS
LIN {X 0.185,Y -687.610,Z 876.422,A 0.000,B 0.000,C 90.000,E1 292.025} C_DIS
LIN {X 0.296,Y -686.792,Z 876.422,A 0.000,B 0.000,C 90.000,E1 291.897} C_DIS
LIN {X 0.148,Y -685.576,Z 876.421,A 0.000,B 0.000,C 90.000,E1 291.791} C_DIS
LIN {X 0.249,Y -681.018,Z 876.419,A 0.000,B 0.000,C 90.000,E1 291.461} C_DIS
LIN {X -0.260,Y -679.438,Z 876.419,A 0.000,B 0.000,C 90.000,E1 291.408} C_DIS
LIN {X 0.113,Y -677.604,Z 876.418,A 0.000,B 0.000,C 90.000,E1 291.280} C_DIS
LIN {X -0.298,Y -670.481,Z 876.417,A 0.000,B 0.000,C 90.000,E1 291.099} C_DIS
LIN {X -0.054,Y -661.381,Z 876.416,A 0.000,B 0.000,C 90.000,E1 290.844} C_DIS
LIN {X -0.244,Y -659.341,Z 876.415,A 0.000,B 0.000,C 90.000,E1 290.791} C_DIS
LIN {X -0.149,Y -653.823,Z 876.414,A 0.000,B 0.000,C 90.000,E1 290.536} C_DIS
LIN {X -0.347,Y -652.497,Z 876.413,A 0.000,B 0.000,C 90.000,E1 290.429} C_DIS
LIN {X 0.222,Y -652.462,Z 876.413,A 0.000,B 0.000,C 90.000,E1 290.375} C_DIS
LIN {X 0.042,Y -652.204,Z 876.413,A 0.000,B 0.000,C 90.000,E1 290.248} C_DIS
LIN {X 0.166,Y -652.334,Z 876.412,A 0.000,B 0.000,C 90.000,E1 290.120} C_DIS
LIN {X 0.029,Y -652.906,Z 876.411,A 0.000,B 0.000,C 90.000,E1 289.885} C_DIS
LIN {X 0.113,Y -653.974,Z 876.409,A 0.000,B 0.000,C 90.000,E1 289.631} C_DIS
LIN {X -0.233,Y -660.962,Z 876.402,A 0.000,B 0.000,C 90.000,E1 288.308} C_DIS
LIN {X -0.332,Y -664.629,Z 876.398,A 0.000,B 0.000,C 90.000,E1 287.583} C_DIS
LIN {X -0.370,Y -666.371,Z 876.396,A 0.000,B 0.000,C 90.000,E1 287.221} C_DIS
LIN {X 0.293,Y -668.453,Z 876.393,A 0.000,B 0.000,C 90.000,E1 286.677} C_DIS
LIN {X 0.069,Y -671.064,Z 876.389,A 0.000,B 0.000,C 90.000,E1 285.969} C_DIS
LIN {X 0.052,Y -673.187,Z 876.385,A 0.000,B 0.000,C 90.000,E1 285.245} C_DIS
LIN {X -0.067,Y -674.356,Z 876.382,A 0.000,B 0.000,C 90.000,E1 284.773} C_DIS
LIN {X -0.232,Y -675.703,Z 876.378,A 0.000,B 0.000,C 90.000,E1 284.064} C_DIS
LIN {X -0.334,Y -676.447,Z 876.375,A 0.000,B 0.000,C 90.000,E1 283.592} C_DIS
LIN {X 0.180,Y -677.264,Z 876.371,A 0.000,B 0.000,C 90.000,E1 282.827} C_DIS
LIN {X 0.041,Y -677.875,Z 876.367,A 0.000,B 0.000,C 90.000,E1 282.119} C_DIS
LIN {X -0.007,Y -678.037,Z 876.366,A 0.000,B 0.000,C 90.000,E1 281.883} C_DIS
LIN {X -0.235,Y -678.115,Z 876.363,A 0.000,B 0.000,C 90.000,E1 281.422} C_DIS
LIN {X 0.290,Y -677.769,Z 876.359,A 0.000,B 0.000,C 90.000,E1 280.658} C_DIS
LIN {X 0.069,Y -677.315,Z 876.357,A 0.000,B 0.000,C 90.000,E1 280.197} C_DIS
LIN {X -0.035,Y -676.579,Z 876.354,A 0.000,B 0.000,C 90.000,E1 279.726} C_DIS
LIN {X -0.259,Y -675.534,Z 876.351,A 0.000,B 0.000,C 90.000,E1 279.265} C_DIS
LIN {X 0.182,Y -674.165,Z 876.349,A 0.000,B 0.000,C 90.000,E1 278.746} C_DIS
LIN {X 0.049,Y -672.502,Z 876.346,A 0.000,B 0.000,C 90.000,E1 278.276} C_DIS
LIN {X -0.119,Y -671.613,Z 876.345,A 0.000,B 0.000,C 90.000,E1 278.049} C_DIS
LIN {X 0.299,Y -669.510,Z 876.342,A 0.000,B 0.000,C 90.000,E1 277.530} C_DIS
LIN {X 0.037,Y -666.490,Z 876.339,A 0.000,B 0.000,C 90.000,E1 276.947} C_DIS
